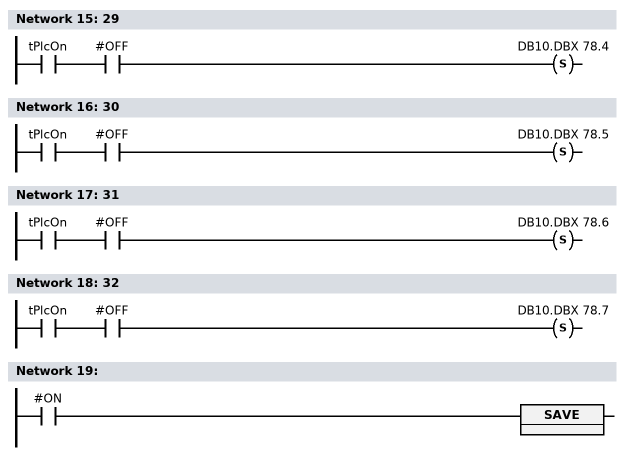
[picture p213: Errors_017-032_GEN2 networks 15-19]
NETWORK
TITLE = 29
      A     "tPlcOn";
      A     #OFF;
      S     DB10.DBX 78.4;
NETWORK
TITLE = 30
      A     "tPlcOn";
      A     #OFF;
      S     DB10.DBX 78.5;
NETWORK
TITLE = 31
      A     "tPlcOn";
      A     #OFF;
      S     DB10.DBX 78.6;
NETWORK
TITLE = 32
      A     "tPlcOn";
      A     #OFF;
      S     DB10.DBX 78.7;
NETWORK
TITLE =
      A     #ON;
      SAVE;
END_FUNCTION

FUNCTION "Errors_033-048_NET" : VOID	// FC 44
TITLE = Errors NET
VERSION : 0.1
VAR_TEMP
  ON : BOOL ;
  OFF : BOOL ;
  tmp_value : INT ;
END_VAR
BEGIN
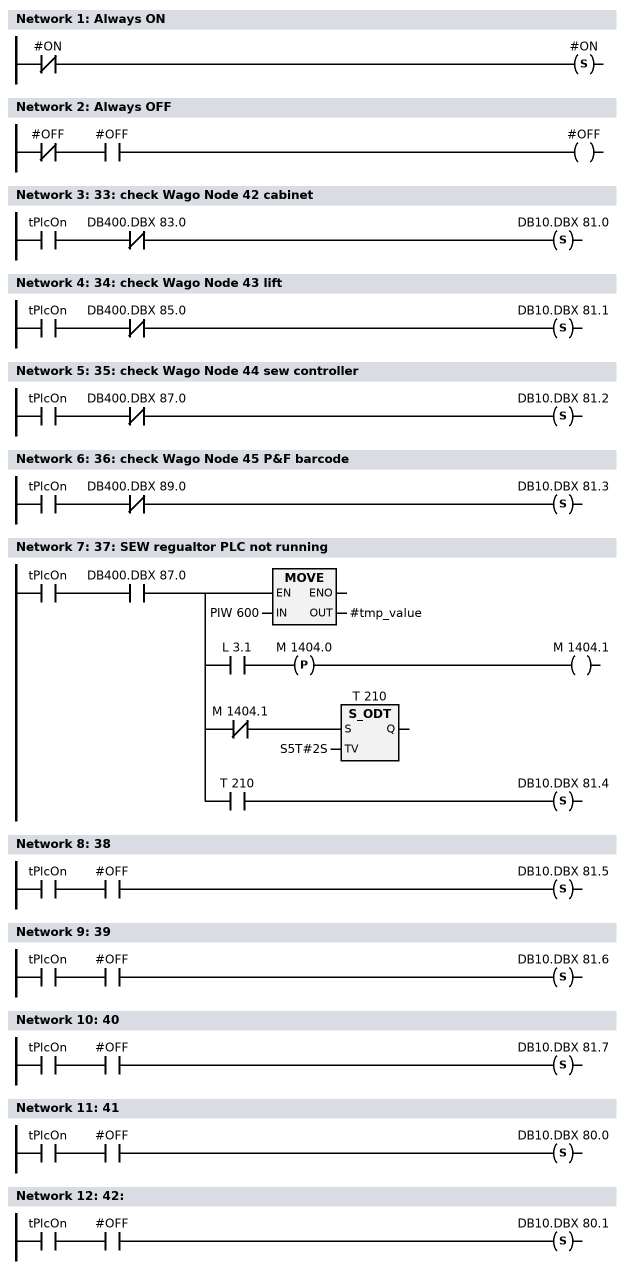
NETWORK
TITLE = Always ON
      AN    #ON;
      S     #ON;
NETWORK
TITLE = Always OFF
      AN    #OFF;
      A     #OFF;
      =     #OFF;
NETWORK
TITLE = 33: check Wago Node 42 cabinet
      A     "tPlcOn";
      AN    DB400.DBX 83.0;
      S     DB10.DBX 81.0;
NETWORK
TITLE = 34: check Wago Node 43 lift
      A     "tPlcOn";
      AN    DB400.DBX 85.0;
      S     DB10.DBX 81.1;
NETWORK
TITLE = 35: check Wago Node 44 sew controller
      A     "tPlcOn";
      AN    DB400.DBX 87.0;
      S     DB10.DBX 81.2;
NETWORK
TITLE = 36: check Wago Node 45 P&F barcode
      A     "tPlcOn";
      AN    DB400.DBX 89.0;
      S     DB10.DBX 81.3;
NETWORK
TITLE = 37: SEW regualtor PLC not running
      A     "tPlcOn";
      A     DB400.DBX 87.0;
      =     L 4.0;
      A     L 4.0;
      JNB   _001;
      L     PIW 600;
      T     #tmp_value;
_001: NOP   0;
      A     L 4.0;
      A     L 3.1;
      FP    M 1404.0;
      =     M 1404.1;
      A     L 4.0;
      AN    M 1404.1;
      L     S5T#2S;
      SD    T 210;
      NOP   0;
      NOP   0;
      NOP   0;
      NOP   0;
      A     L 4.0;
      A     T 210;
      S     DB10.DBX 81.4;
NETWORK
TITLE = 38
      A     "tPlcOn";
      A     #OFF;
      S     DB10.DBX 81.5;
NETWORK
TITLE = 39
      A     "tPlcOn";
      A     #OFF;
      S     DB10.DBX 81.6;
NETWORK
TITLE = 40
      A     "tPlcOn";
      A     #OFF;
      S     DB10.DBX 81.7;
NETWORK
TITLE = 41
      A     "tPlcOn";
      A     #OFF;
      S     DB10.DBX 80.0;
NETWORK
TITLE = 42:
      A     "tPlcOn";
      A     #OFF;
      S     DB10.DBX 80.1;
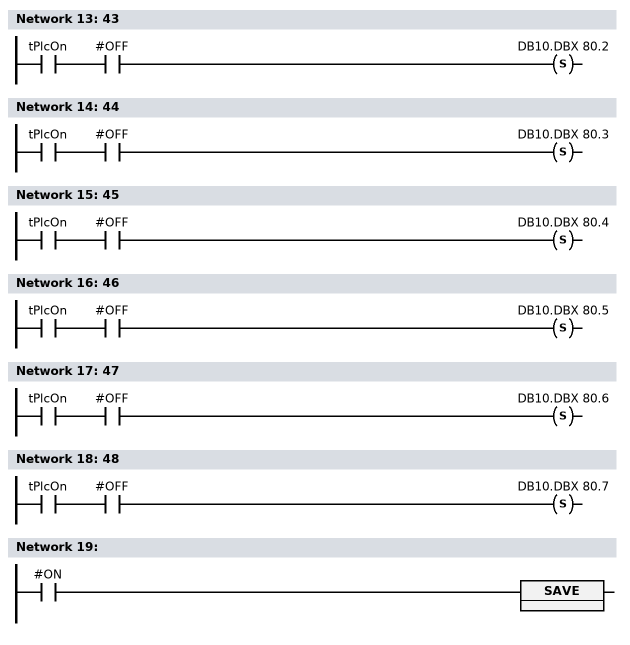
NETWORK
TITLE = 43
      A     "tPlcOn";
      A     #OFF;
      S     DB10.DBX 80.2;
NETWORK
TITLE = 44
      A     "tPlcOn";
      A     #OFF;
      S     DB10.DBX 80.3;
NETWORK
TITLE = 45
      A     "tPlcOn";
      A     #OFF;
      S     DB10.DBX 80.4;
NETWORK
TITLE = 46
      A     "tPlcOn";
      A     #OFF;
      S     DB10.DBX 80.5;
NETWORK
TITLE = 47
      A     "tPlcOn";
      A     #OFF;
      S     DB10.DBX 80.6;
NETWORK
TITLE = 48
      A     "tPlcOn";
      A     #OFF;
      S     DB10.DBX 80.7;
NETWORK
TITLE =
      A     #ON;
      SAVE;
END_FUNCTION

FUNCTION "Errors_113-128" : VOID	// FC 45
TITLE = Errors 113 - 128
VERSION : 0.1
VAR_TEMP
  ON : BOOL ;
END_VAR
BEGIN
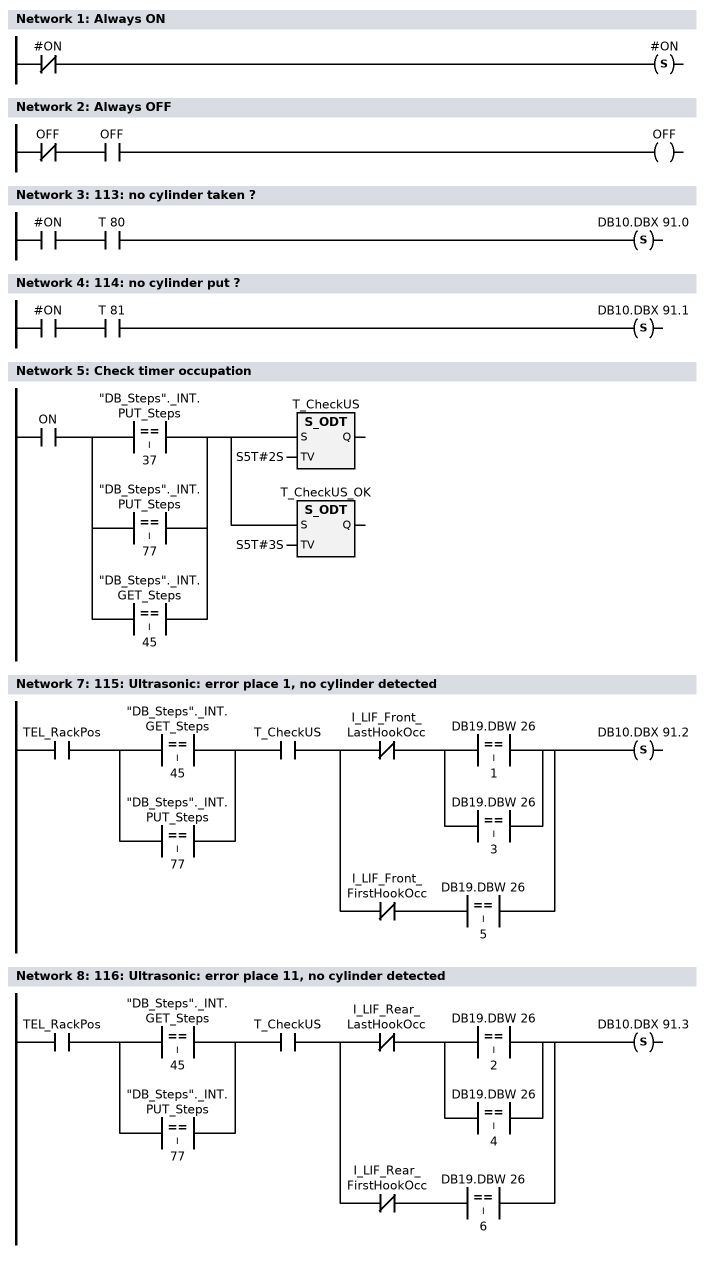
NETWORK
TITLE = Always ON
      AN    #ON;
      S     #ON;
NETWORK
TITLE = Always OFF
      AN    "OFF";
      A     "OFF";
      =     "OFF";
NETWORK
TITLE = 113: no cylinder taken ?
      A     #ON;
      A     T 80;
      S     DB10.DBX 91.0;
NETWORK
TITLE = 114: no cylinder put ?
      A     #ON;
      A     T 81;
      S     DB10.DBX 91.1;
NETWORK
TITLE = Check timer occupation
//T160 time to error
//T161 time to cont
      A     "ON";
      A(;
      O(;
      L     "DB_Steps"._INT.PUT_Steps;
      L     37;
      ==I;
      );
      O(;
      L     "DB_Steps"._INT.PUT_Steps;
      L     77;
      ==I;
      );
      O(;
      L     "DB_Steps"._INT.GET_Steps;
      L     45;
      ==I;
      );
      );
      =     L 1.0;
      A     L 1.0;
      L     S5T#2S;
      SD    "T_CheckUS";
      NOP   0;
      NOP   0;
      NOP   0;
      NOP   0;
      A     L 1.0;
      L     S5T#3S;
      SD    "T_CheckUS_OK";
      NOP   0;
      NOP   0;
      NOP   0;
      NOP   0;
NETWORK
TITLE =
NETWORK
TITLE = 115: Ultrasonic: error place 1, no cylinder detected
      A     "TEL_RackPos";
      A(;
      O(;
      L     "DB_Steps"._INT.GET_Steps;
      L     45;
      ==I;
      );
      O(;
      L     "DB_Steps"._INT.PUT_Steps;
      L     77;
      ==I;
      );
      );
      A     "T_CheckUS";
      A(;
      AN    "I_LIF_Front_LastHookOcc";
      A(;
      O(;
      L     DB19.DBW 26;
      L     1;
      ==I;
      );
      O(;
      L     DB19.DBW 26;
      L     3;
      ==I;
      );
      );
      O;
      AN    "I_LIF_Front_FirstHookOcc";
      A(;
      L     DB19.DBW 26;
      L     5;
      ==I;
      );
      );
      S     DB10.DBX 91.2;
NETWORK
TITLE = 116: Ultrasonic: error place 11, no cylinder detected
      A     "TEL_RackPos";
      A(;
      O(;
      L     "DB_Steps"._INT.GET_Steps;
      L     45;
      ==I;
      );
      O(;
      L     "DB_Steps"._INT.PUT_Steps;
      L     77;
      ==I;
      );
      );
      A     "T_CheckUS";
      A(;
      AN    "I_LIF_Rear_LastHookOcc";
      A(;
      O(;
      L     DB19.DBW 26;
      L     2;
      ==I;
      );
      O(;
      L     DB19.DBW 26;
      L     4;
      ==I;
      );
      );
      O;
      AN    "I_LIF_Rear_FirstHookOcc";
      A(;
      L     DB19.DBW 26;
      L     6;
      ==I;
      );
      );
      S     DB10.DBX 91.3;
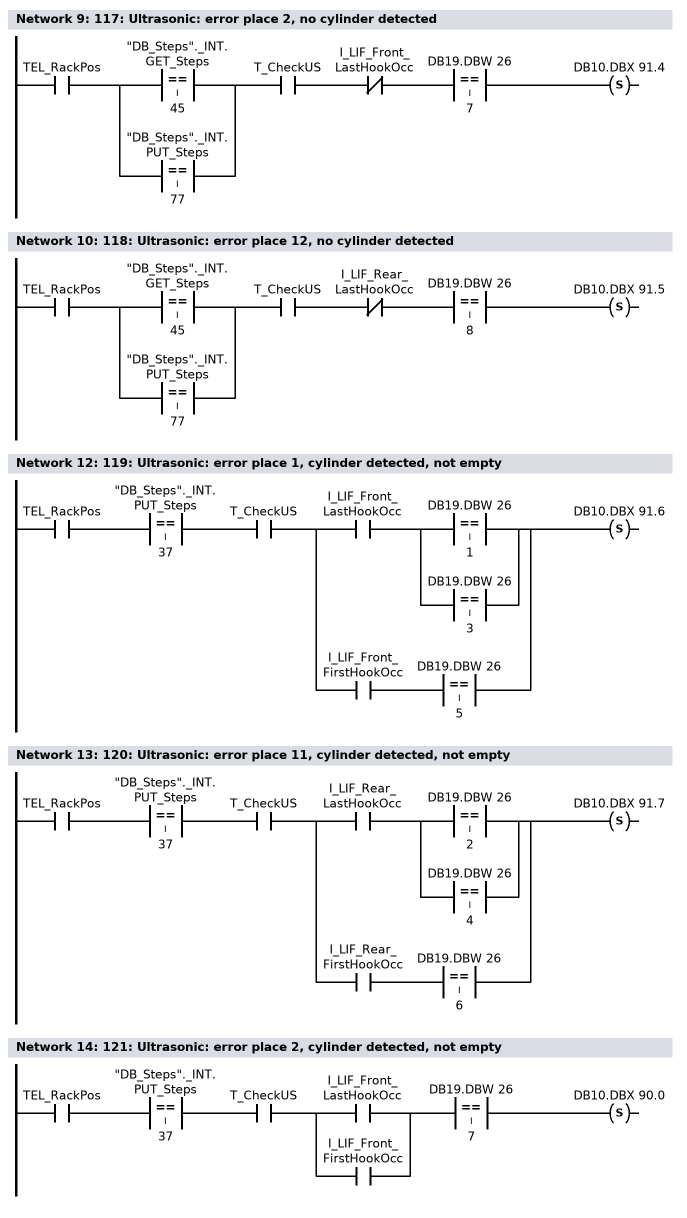
NETWORK
TITLE = 117: Ultrasonic: error place 2, no cylinder detected
      A     "TEL_RackPos";
      A(;
      O(;
      L     "DB_Steps"._INT.GET_Steps;
      L     45;
      ==I;
      );
      O(;
      L     "DB_Steps"._INT.PUT_Steps;
      L     77;
      ==I;
      );
      );
      A     "T_CheckUS";
      AN    "I_LIF_Front_LastHookOcc";
      A(;
      L     DB19.DBW 26;
      L     7;
      ==I;
      );
      S     DB10.DBX 91.4;
NETWORK
TITLE = 118: Ultrasonic: error place 12, no cylinder detected
      A     "TEL_RackPos";
      A(;
      O(;
      L     "DB_Steps"._INT.GET_Steps;
      L     45;
      ==I;
      );
      O(;
      L     "DB_Steps"._INT.PUT_Steps;
      L     77;
      ==I;
      );
      );
      A     "T_CheckUS";
      AN    "I_LIF_Rear_LastHookOcc";
      A(;
      L     DB19.DBW 26;
      L     8;
      ==I;
      );
      S     DB10.DBX 91.5;
NETWORK
TITLE =
NETWORK
TITLE = 119: Ultrasonic: error place 1, cylinder detected, not empty
      A     "TEL_RackPos";
      A(;
      L     "DB_Steps"._INT.PUT_Steps;
      L     37;
      ==I;
      );
      A     "T_CheckUS";
      A(;
      A     "I_LIF_Front_LastHookOcc";
      A(;
      O(;
      L     DB19.DBW 26;
      L     1;
      ==I;
      );
      O(;
      L     DB19.DBW 26;
      L     3;
      ==I;
      );
      );
      O;
      A     "I_LIF_Front_FirstHookOcc";
      A(;
      L     DB19.DBW 26;
      L     5;
      ==I;
      );
      );
      S     DB10.DBX 91.6;
NETWORK
TITLE = 120: Ultrasonic: error place 11, cylinder detected, not empty
      A     "TEL_RackPos";
      A(;
      L     "DB_Steps"._INT.PUT_Steps;
      L     37;
      ==I;
      );
      A     "T_CheckUS";
      A(;
      A     "I_LIF_Rear_LastHookOcc";
      A(;
      O(;
      L     DB19.DBW 26;
      L     2;
      ==I;
      );
      O(;
      L     DB19.DBW 26;
      L     4;
      ==I;
      );
      );
      O;
      A     "I_LIF_Rear_FirstHookOcc";
      A(;
      L     DB19.DBW 26;
      L     6;
      ==I;
      );
      );
      S     DB10.DBX 91.7;
NETWORK
TITLE = 121: Ultrasonic: error place 2, cylinder detected, not empty
      A     "TEL_RackPos";
      A(;
      L     "DB_Steps"._INT.PUT_Steps;
      L     37;
      ==I;
      );
      A     "T_CheckUS";
      A(;
      O     "I_LIF_Front_LastHookOcc";
      O     "I_LIF_Front_FirstHookOcc";
      );
      A(;
      L     DB19.DBW 26;
      L     7;
      ==I;
      );
      S     DB10.DBX 90.0;
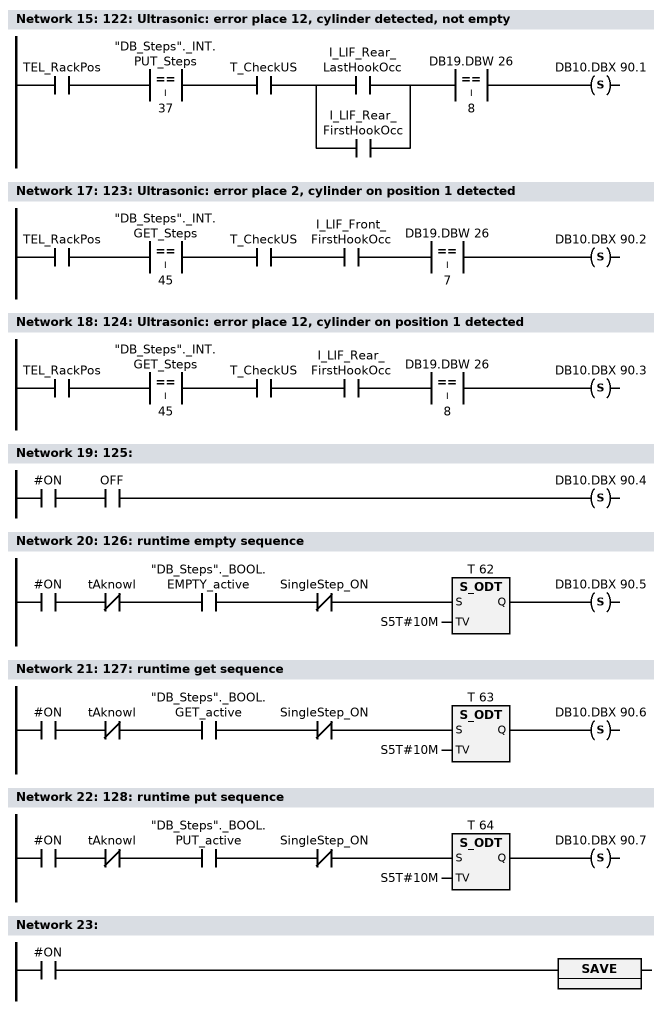
NETWORK
TITLE = 122: Ultrasonic: error place 12, cylinder detected, not empty
      A     "TEL_RackPos";
      A(;
      L     "DB_Steps"._INT.PUT_Steps;
      L     37;
      ==I;
      );
      A     "T_CheckUS";
      A(;
      O     "I_LIF_Rear_LastHookOcc";
      O     "I_LIF_Rear_FirstHookOcc";
      );
      A(;
      L     DB19.DBW 26;
      L     8;
      ==I;
      );
      S     DB10.DBX 90.1;
NETWORK
TITLE =
NETWORK
TITLE = 123: Ultrasonic: error place 2, cylinder on position 1 detected
      A     "TEL_RackPos";
      A(;
      L     "DB_Steps"._INT.GET_Steps;
      L     45;
      ==I;
      );
      A     "T_CheckUS";
      A     "I_LIF_Front_FirstHookOcc";
      A(;
      L     DB19.DBW 26;
      L     7;
      ==I;
      );
      S     DB10.DBX 90.2;
NETWORK
TITLE = 124: Ultrasonic: error place 12, cylinder on position 1 detected
      A     "TEL_RackPos";
      A(;
      L     "DB_Steps"._INT.GET_Steps;
      L     45;
      ==I;
      );
      A     "T_CheckUS";
      A     "I_LIF_Rear_FirstHookOcc";
      A(;
      L     DB19.DBW 26;
      L     8;
      ==I;
      );
      S     DB10.DBX 90.3;
NETWORK
TITLE = 125:
      A     #ON;
      A     "OFF";
      S     DB10.DBX 90.4;
NETWORK
TITLE = 126: runtime empty sequence
      A     #ON;
      AN    "tAknowl";
      A     "DB_Steps"._BOOL.EMPTY_active;
      AN    "SingleStep_ON";
      L     S5T#10M;
      SD    T 62;
      NOP   0;
      NOP   0;
      NOP   0;
      A     T 62;
      S     DB10.DBX 90.5;
NETWORK
TITLE = 127: runtime get sequence
      A     #ON;
      AN    "tAknowl";
      A     "DB_Steps"._BOOL.GET_active;
      AN    "SingleStep_ON";
      L     S5T#10M;
      SD    T 63;
      NOP   0;
      NOP   0;
      NOP   0;
      A     T 63;
      S     DB10.DBX 90.6;
NETWORK
TITLE = 128: runtime put sequence
      A     #ON;
      AN    "tAknowl";
      A     "DB_Steps"._BOOL.PUT_active;
      AN    "SingleStep_ON";
      L     S5T#10M;
      SD    T 64;
      NOP   0;
      NOP   0;
      NOP   0;
      A     T 64;
      S     DB10.DBX 90.7;
NETWORK
TITLE =
      A     #ON;
      SAVE;
END_FUNCTION

FUNCTION "Errors_129-144_08" : VOID	// FC 46
TITLE = Errors
VERSION : 0.1
VAR_TEMP
  ON : BOOL ;
  OFF : BOOL ;
END_VAR
BEGIN
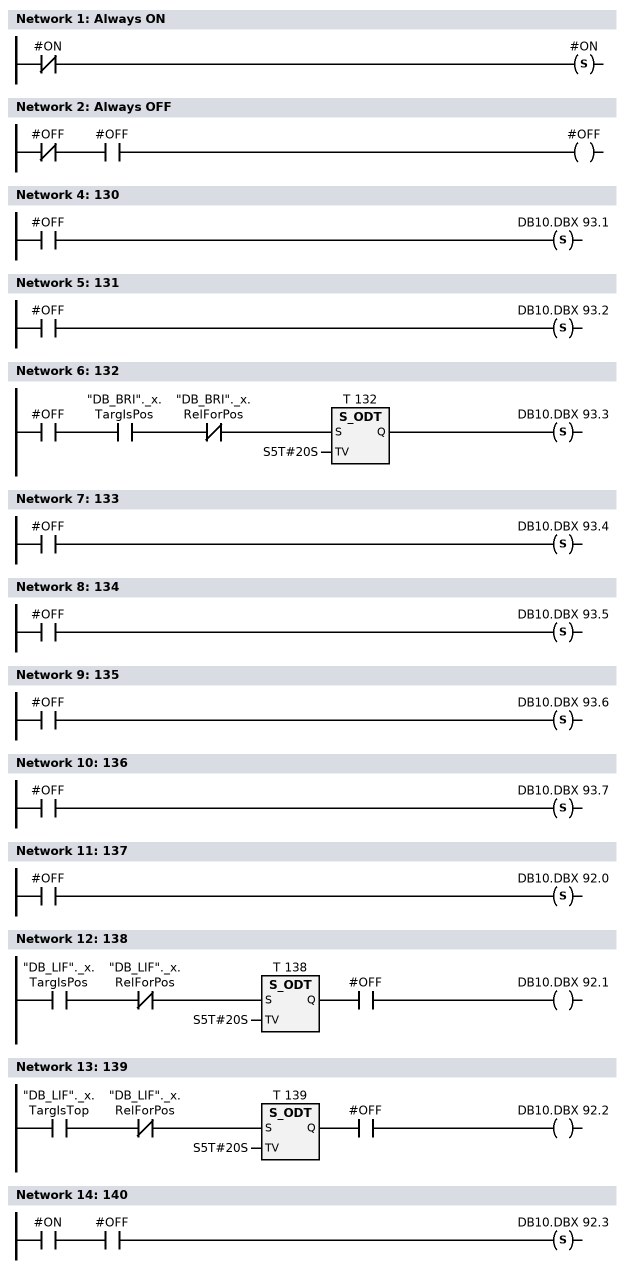
NETWORK
TITLE = Always ON
      AN    #ON;
      S     #ON;
NETWORK
TITLE = Always OFF
      AN    #OFF;
      A     #OFF;
      =     #OFF;
NETWORK
TITLE = 129
//00 in Steps_PUT/NW65
NETWORK
TITLE = 130
//01
      A     #OFF;
      S     DB10.DBX 93.1;
NETWORK
TITLE = 131
//02
      A     #OFF;
      S     DB10.DBX 93.2;
NETWORK
TITLE = 132
//Brücke keine Freigabe für Positionierung
      A     #OFF;
      A     "DB_BRI"._x.TargIsPos;
      AN    "DB_BRI"._x.RelForPos;
      L     S5T#20S;
      SD    T 132;
      NOP   0;
      NOP   0;
      NOP   0;
      A     T 132;
      S     DB10.DBX 93.3;
NETWORK
TITLE = 133
//04
      A     #OFF;
      S     DB10.DBX 93.4;
NETWORK
TITLE = 134
//05
      A     #OFF;
      S     DB10.DBX 93.5;
NETWORK
TITLE = 135
//06
      A     #OFF;
      S     DB10.DBX 93.6;
NETWORK
TITLE = 136
//07
      A     #OFF;
      S     DB10.DBX 93.7;
NETWORK
TITLE = 137
//08
      A     #OFF;
      S     DB10.DBX 92.0;
NETWORK
TITLE = 138
//Lift keine Freigabe für Positionierung
      A(;
      A     "DB_LIF"._x.TargIsPos;
      AN    "DB_LIF"._x.RelForPos;
      L     S5T#20S;
      SD    T 138;
      NOP   0;
      NOP   0;
      NOP   0;
      A     T 138;
      );
      A     #OFF;
      =     DB10.DBX 92.1;
NETWORK
TITLE = 139
//Lift keine Freigabe für Positionierung
      A(;
      A     "DB_LIF"._x.TargIsTop;
      AN    "DB_LIF"._x.RelForPos;
      L     S5T#20S;
      SD    T 139;
      NOP   0;
      NOP   0;
      NOP   0;
      A     T 139;
      );
      A     #OFF;
      =     DB10.DBX 92.2;
NETWORK
TITLE = 140
//Messung Umfang nicht erfolgreich
      A     #ON;
      A     #OFF;
      S     DB10.DBX 92.3;
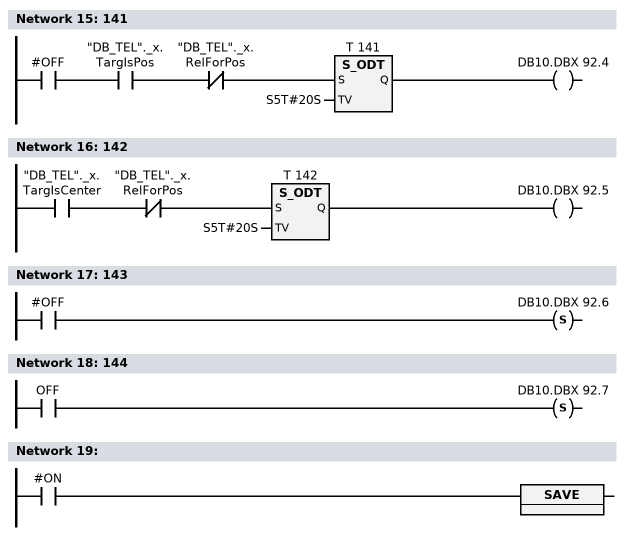
NETWORK
TITLE = 141
//Teleskope keine Freigabe für Positionierung
      A     #OFF;
      A     "DB_TEL"._x.TargIsPos;
      AN    "DB_TEL"._x.RelForPos;
      L     S5T#20S;
      SD    T 141;
      NOP   0;
      NOP   0;
      NOP   0;
      A     T 141;
      =     DB10.DBX 92.4;
NETWORK
TITLE = 142
//Teleskope keine Freigabe für Positionierung
      A     "DB_TEL"._x.TargIsCenter;
      AN    "DB_TEL"._x.RelForPos;
      L     S5T#20S;
      SD    T 142;
      NOP   0;
      NOP   0;
      NOP   0;
      A     T 142;
      =     DB10.DBX 92.5;
NETWORK
TITLE = 143
      A     #OFF;
      S     DB10.DBX 92.6;
NETWORK
TITLE = 144
      A     "OFF";
      S     DB10.DBX 92.7;
NETWORK
TITLE =
      A     #ON;
      SAVE;
END_FUNCTION

FUNCTION "Errors_145-160" : VOID	// FC 47
TITLE = Messages 145 - 160
VERSION : 0.1
VAR_TEMP
  ON : BOOL ;
  OFF : BOOL ;
END_VAR
BEGIN
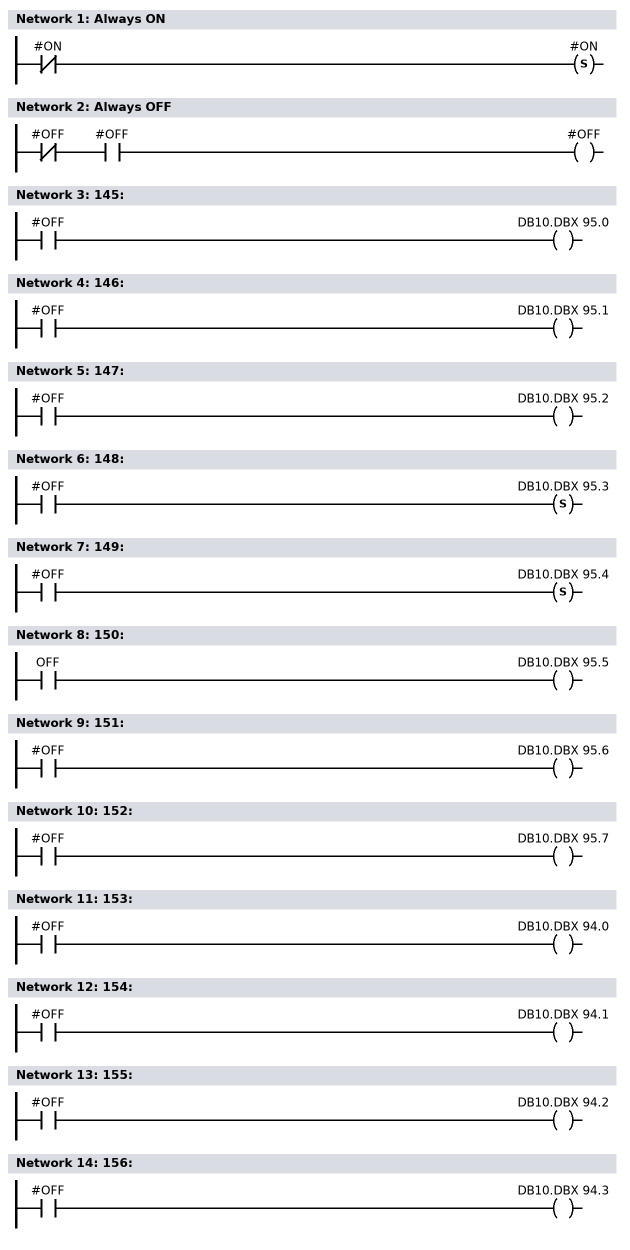
NETWORK
TITLE = Always ON
      AN    #ON;
      S     #ON;
NETWORK
TITLE = Always OFF
      AN    #OFF;
      A     #OFF;
      =     #OFF;
NETWORK
TITLE = 145:
//keine Freigabe Teleskop Fach 1 (Fachtyp)
      A     #OFF;
      =     DB10.DBX 95.0;
NETWORK
TITLE = 146:
//keine Freigabe Teleskop Fach 2 (Fachtyp)
      A     #OFF;
      =     DB10.DBX 95.1;
NETWORK
TITLE = 147:
//keine Freigabe Teleskop Ladestation 1
      A     #OFF;
      =     DB10.DBX 95.2;
NETWORK
TITLE = 148:
//keine Freigabe Teleskop Ladestation 2
      A     #OFF;
      S     DB10.DBX 95.3;
NETWORK
TITLE = 149:
//keine Freigabe Teleskop Ladestation 3
      A     #OFF;
      S     DB10.DBX 95.4;
NETWORK
TITLE = 150:
      A     "OFF";
      =     DB10.DBX 95.5;
NETWORK
TITLE = 151:
      A     #OFF;
      =     DB10.DBX 95.6;
NETWORK
TITLE = 152:
      A     #OFF;
      =     DB10.DBX 95.7;
NETWORK
TITLE = 153:
      A     #OFF;
      =     DB10.DBX 94.0;
NETWORK
TITLE = 154:
      A     #OFF;
      =     DB10.DBX 94.1;
NETWORK
TITLE = 155:
      A     #OFF;
      =     DB10.DBX 94.2;
NETWORK
TITLE = 156:
      A     #OFF;
      =     DB10.DBX 94.3;
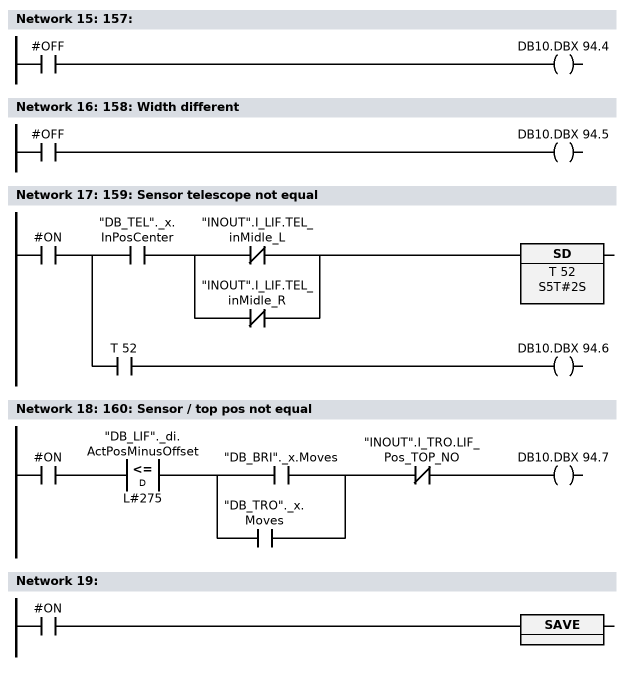
NETWORK
TITLE = 157:
      A     #OFF;
      =     DB10.DBX 94.4;
NETWORK
TITLE = 158: Width different
      A     #OFF;
      =     DB10.DBX 94.5;
NETWORK
TITLE = 159: Sensor telescope not equal
      A     #ON;
      =     L 1.0;
      A     L 1.0;
      A     "DB_TEL"._x.InPosCenter;
      A(;
      ON    "INOUT".I_LIF.TEL_inMidle_L;
      ON    "INOUT".I_LIF.TEL_inMidle_R;
      );
      L     S5T#2S;
      SD    T 52;
      A     L 1.0;
      A     T 52;
      =     DB10.DBX 94.6;
NETWORK
TITLE = 160: Sensor / top pos not equal
      A     #ON;
      A(;
      L     "DB_LIF"._di.ActPosMinusOffset;
      L     L#275;
      <=D;
      );
      A(;
      O     "DB_BRI"._x.Moves;
      O     "DB_TRO"._x.Moves;
      );
      AN    "INOUT".I_TRO.LIF_Pos_TOP_NO;
      =     DB10.DBX 94.7;
NETWORK
TITLE =
      A     #ON;
      SAVE;
END_FUNCTION

FUNCTION "EOff_MachineOff" : VOID	// FC 48
TITLE = EOff Machine off
//TODO disable the remote in auto
VERSION : 0.1
VAR_TEMP
  INT_DivEoff : BOOL ;
  INT_Err_GEN1 : BOOL ;
  INT_Err_GEN2 : BOOL ;
  INT_Err_NET : BOOL ;
  INT_Err_BRI : BOOL ;
  INT_Err_TRO : BOOL ;
  INT_Err_LIF : BOOL ;
  INT_Err_TEL : BOOL ;
  INT_Warn : BOOL ;
  INT_OPM1 : BOOL ;
  INT_OPM2 : BOOL ;
  INT_ERR_06 : BOOL ;
  INT_ERR_07 : BOOL ;
  INT_ERR_08 : BOOL ;
  INT_ERR_09 : BOOL ;
  INT_ERR_10 : BOOL ;
  INT_ERR_11 : BOOL ;
  INT_MSG_01 : BOOL ;
  INT_MSG_02 : BOOL ;
  INT_MSG_03 : BOOL ;
  INT_MSG_04 : BOOL ;
  ON : BOOL ;
  OFF : BOOL ;
END_VAR
BEGIN
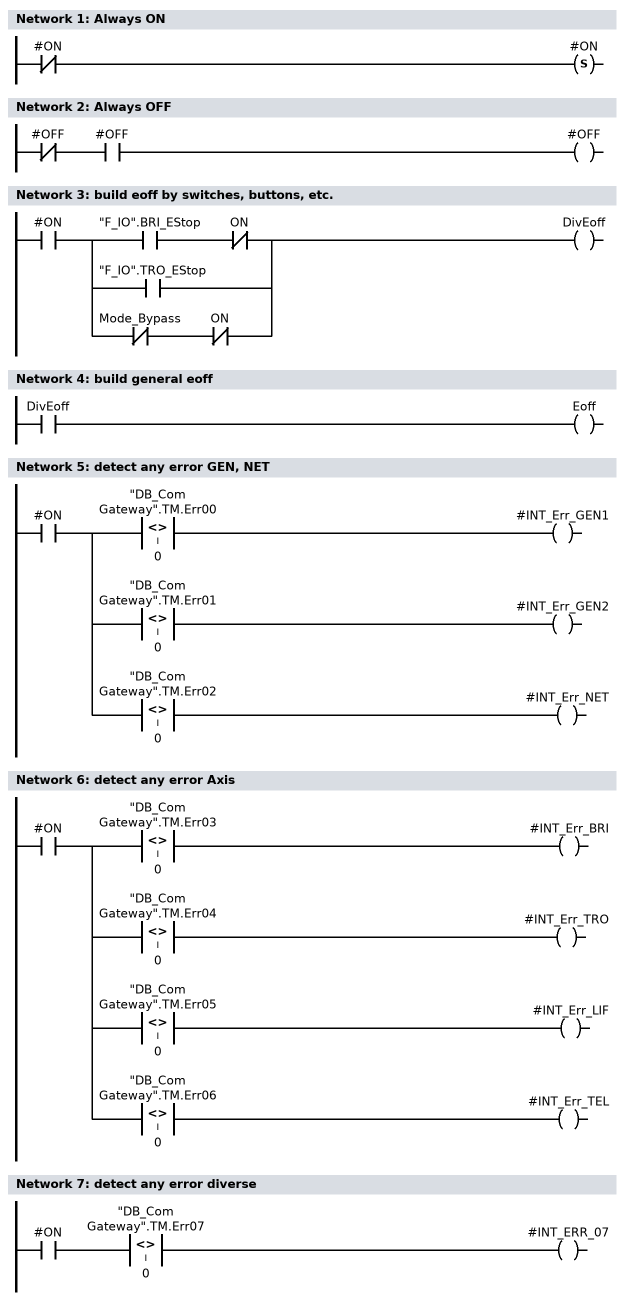
NETWORK
TITLE = Always ON
      AN    #ON;
      S     #ON;
NETWORK
TITLE = Always OFF
      AN    #OFF;
      A     #OFF;
      =     #OFF;
NETWORK
TITLE = build eoff by switches, buttons, etc.
      A     #ON;
      A(;
      A     "F_IO".BRI_EStop;
      AN    "ON";
      O     "F_IO".TRO_EStop;
      O;
      AN    "Mode_Bypass";
      AN    "ON";
      );
      =     "DivEoff";
NETWORK
TITLE = build general eoff
      A     "DivEoff";
      =     "Eoff";
NETWORK
TITLE = detect any error GEN, NET
      A     #ON;
      =     L 3.0;
      A     L 3.0;
      A(;
      L     "DB_ComGateway".TM.Err00;
      L     0;
      <>I;
      );
      =     #INT_Err_GEN1;
      A     L 3.0;
      A(;
      L     "DB_ComGateway".TM.Err01;
      L     0;
      <>I;
      );
      =     #INT_Err_GEN2;
      A     L 3.0;
      A(;
      L     "DB_ComGateway".TM.Err02;
      L     0;
      <>I;
      );
      =     #INT_Err_NET;
NETWORK
TITLE = detect any error Axis
      A     #ON;
      =     L 3.0;
      A     L 3.0;
      A(;
      L     "DB_ComGateway".TM.Err03;
      L     0;
      <>I;
      );
      =     #INT_Err_BRI;
      A     L 3.0;
      A(;
      L     "DB_ComGateway".TM.Err04;
      L     0;
      <>I;
      );
      =     #INT_Err_TRO;
      A     L 3.0;
      A(;
      L     "DB_ComGateway".TM.Err05;
      L     0;
      <>I;
      );
      =     #INT_Err_LIF;
      A     L 3.0;
      A(;
      L     "DB_ComGateway".TM.Err06;
      L     0;
      <>I;
      );
      =     #INT_Err_TEL;
NETWORK
TITLE = detect any error diverse
      A     #ON;
      A(;
      L     "DB_ComGateway".TM.Err07;
      L     0;
      <>I;
      );
      =     #INT_ERR_07;
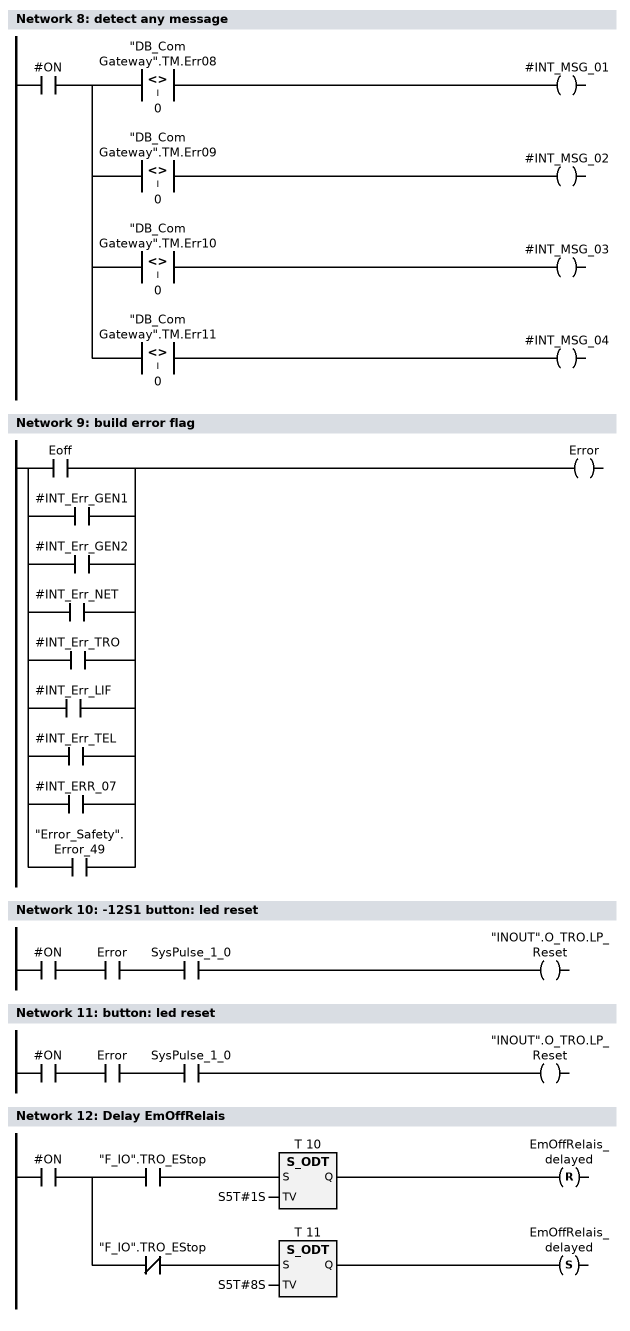
NETWORK
TITLE = detect any message
      A     #ON;
      =     L 3.0;
      A     L 3.0;
      A(;
      L     "DB_ComGateway".TM.Err08;
      L     0;
      <>I;
      );
      =     #INT_MSG_01;
      A     L 3.0;
      A(;
      L     "DB_ComGateway".TM.Err09;
      L     0;
      <>I;
      );
      =     #INT_MSG_02;
      A     L 3.0;
      A(;
      L     "DB_ComGateway".TM.Err10;
      L     0;
      <>I;
      );
      =     #INT_MSG_03;
      A     L 3.0;
      A(;
      L     "DB_ComGateway".TM.Err11;
      L     0;
      <>I;
      );
      =     #INT_MSG_04;
NETWORK
TITLE = build error flag
//xOff for error words
//
      O     "Eoff";
      O     #INT_Err_GEN1;
      O     #INT_Err_GEN2;
      O     #INT_Err_NET;
      O     #INT_Err_TRO;
      O     #INT_Err_LIF;
      O     #INT_Err_TEL;
      O     #INT_ERR_07;
      O     "Error_Safety".Error_49;
      =     "Error";
NETWORK
TITLE = -12S1 button: led reset
      A     #ON;
      A     "Error";
      A     "SysPulse_1_0";
      =     "INOUT".O_TRO.LP_Reset;
NETWORK
TITLE = button: led reset
      A     #ON;
      A     "Error";
      A     "SysPulse_1_0";
      =     "INOUT".O_TRO.LP_Reset;
NETWORK
TITLE = Delay EmOffRelais
      A     #ON;
      =     L 3.0;
      A     L 3.0;
      A     "F_IO".TRO_EStop;
      L     S5T#1S;
      SD    T 10;
      NOP   0;
      NOP   0;
      NOP   0;
      A     T 10;
      R     "EmOffRelais_delayed";
      A     L 3.0;
      AN    "F_IO".TRO_EStop;
      L     S5T#8S;
      SD    T 11;
      NOP   0;
      NOP   0;
      NOP   0;
      A     T 11;
      S     "EmOffRelais_delayed";
END_FUNCTION

FUNCTION "OP_Mode" : VOID	// FC 49
TITLE = OP Mode
//Sicherheitsbaugruppen noch nicht in Betrieb !!!
VERSION : 0.1
VAR_TEMP
  TEMP_DINT_00 : DINT ;
  TEMP_DINT_01 : DINT ;
  TEMP_BOOL_00 : BOOL ;
  TEMP_BOOL_01 : BOOL ;
  TEMP_BOOL_02 : BOOL ;
  TEMP_BOOL_03 : BOOL ;
  TEMP_BOOL_04 : BOOL ;
  TEMP_BOOL_05 : BOOL ;
  TEMP_BOOL_06 : BOOL ;
  value : INT ;
  lampPrio : INT ;
  ON : BOOL ;
  OFF : BOOL ;
  delay : BOOL ;
END_VAR
BEGIN
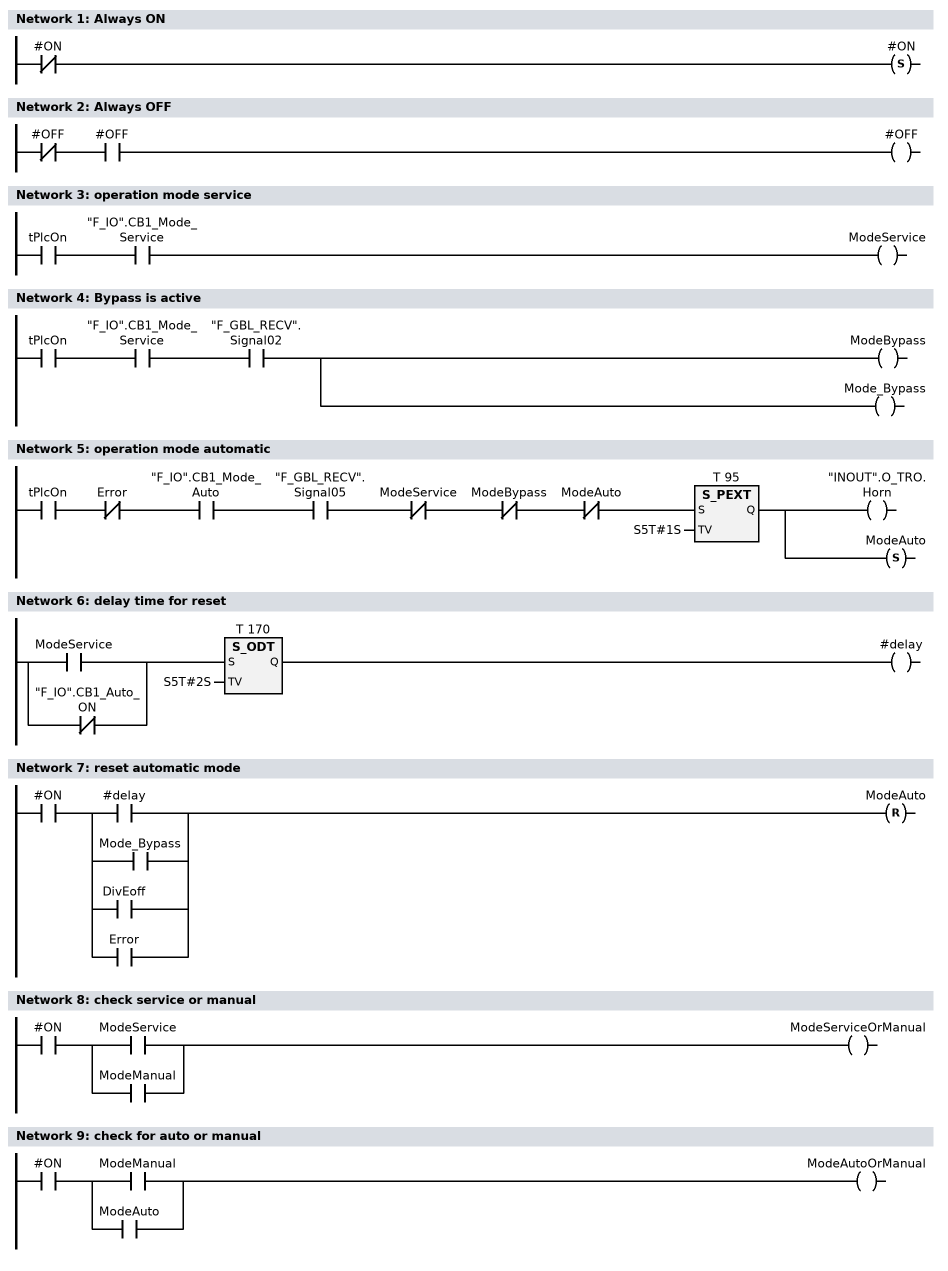
NETWORK
TITLE = Always ON
      AN    #ON;
      S     #ON;
NETWORK
TITLE = Always OFF
      AN    #OFF;
      A     #OFF;
      =     #OFF;
NETWORK
TITLE = operation mode service
      A     "tPlcOn";
      A     "F_IO".CB1_Mode_Service;
      =     "ModeService";
NETWORK
TITLE = Bypass is active
      A     "tPlcOn";
      A     "F_IO".CB1_Mode_Service;
      A     "F_GBL_RECV".Signal02;
      =     "ModeBypass";
      =     "Mode_Bypass";
NETWORK
TITLE = operation mode automatic
      A     "tPlcOn";
      AN    "Error";
      A     "F_IO".CB1_Mode_Auto;
      A     "F_GBL_RECV".Signal05;
      AN    "ModeService";
      AN    "ModeBypass";
      AN    "ModeAuto";
      L     S5T#1S;
      SE    T 95;
      NOP   0;
      NOP   0;
      NOP   0;
      A     T 95;
      =     "INOUT".O_TRO.Horn;
      S     "ModeAuto";
NETWORK
TITLE = delay time for reset
      A(;
      O     "ModeService";
      ON    "F_IO".CB1_Auto_ON;
      );
      L     S5T#2S;
      SD    T 170;
      NOP   0;
      NOP   0;
      NOP   0;
      A     T 170;
      =     #delay;
NETWORK
TITLE = reset automatic mode
      A     #ON;
      A(;
      O     #delay;
      O     "Mode_Bypass";
      O     "DivEoff";
      O     "Error";
      );
      R     "ModeAuto";
NETWORK
TITLE = check service or manual
      A     #ON;
      A(;
      O     "ModeService";
      O     "ModeManual";
      );
      =     "ModeServiceOrManual";
NETWORK
TITLE = check for auto or manual
      A     #ON;
      A(;
      O     "ModeManual";
      O     "ModeAuto";
      );
      =     "ModeAutoOrManual";
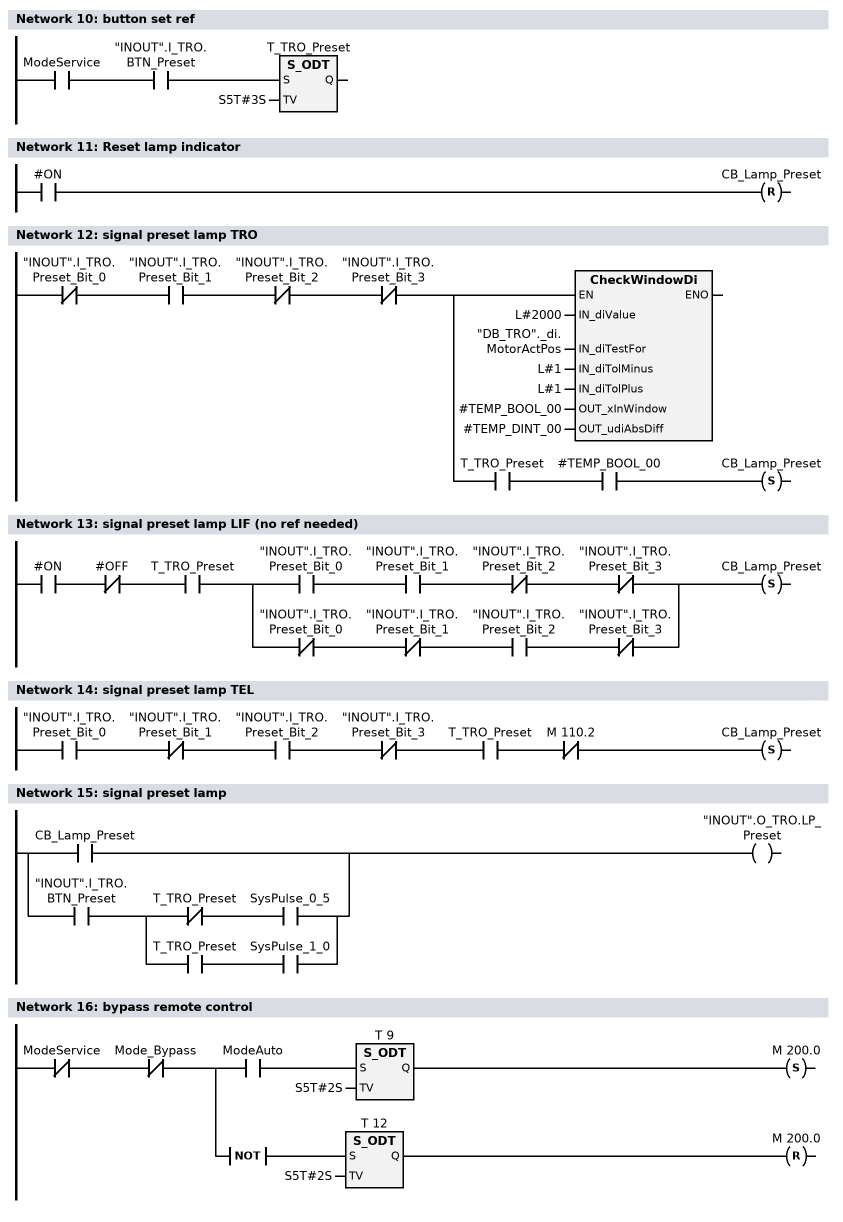
NETWORK
TITLE = button set ref
      A     "ModeService";
      A     "INOUT".I_TRO.BTN_Preset;
      L     S5T#3S;
      SD    "T_TRO_Preset";
      NOP   0;
      NOP   0;
      NOP   0;
      NOP   0;
NETWORK
TITLE = Reset lamp indicator
      A     #ON;
      R     "CB_Lamp_Preset";
NETWORK
TITLE = signal preset lamp TRO
      AN    "INOUT".I_TRO.Preset_Bit_0;
      A     "INOUT".I_TRO.Preset_Bit_1;
      AN    "INOUT".I_TRO.Preset_Bit_2;
      AN    "INOUT".I_TRO.Preset_Bit_3;
      =     L 15.0;
      A     L 15.0;
      JNB   _001;
      CALL  "CheckWindowDi" (
           IN_diValue               := L#2000,
           IN_diTestFor             := "DB_TRO"._di.MotorActPos,
           IN_diTolMinus            := L#1,
           IN_diTolPlus             := L#1,
           OUT_xInWindow            := #TEMP_BOOL_00,
           OUT_udiAbsDiff           := #TEMP_DINT_00);
_001: NOP   0;
      A     L 15.0;
      A     "T_TRO_Preset";
      A     #TEMP_BOOL_00;
      S     "CB_Lamp_Preset";
NETWORK
TITLE = signal preset lamp LIF (no ref needed)
      A     #ON;
      AN    #OFF;
      A     "T_TRO_Preset";
      A(;
      A     "INOUT".I_TRO.Preset_Bit_0;
      A     "INOUT".I_TRO.Preset_Bit_1;
      AN    "INOUT".I_TRO.Preset_Bit_2;
      AN    "INOUT".I_TRO.Preset_Bit_3;
      O;
      AN    "INOUT".I_TRO.Preset_Bit_0;
      AN    "INOUT".I_TRO.Preset_Bit_1;
      A     "INOUT".I_TRO.Preset_Bit_2;
      AN    "INOUT".I_TRO.Preset_Bit_3;
      );
      S     "CB_Lamp_Preset";
NETWORK
TITLE = signal preset lamp TEL
      A     "INOUT".I_TRO.Preset_Bit_0;
      AN    "INOUT".I_TRO.Preset_Bit_1;
      A     "INOUT".I_TRO.Preset_Bit_2;
      AN    "INOUT".I_TRO.Preset_Bit_3;
      A     "T_TRO_Preset";
      AN    M 110.2;
      S     "CB_Lamp_Preset";
NETWORK
TITLE = signal preset lamp
      O     "CB_Lamp_Preset";
      O;
      A     "INOUT".I_TRO.BTN_Preset;
      A(;
      AN    "T_TRO_Preset";
      A     "SysPulse_0_5";
      O;
      A     "T_TRO_Preset";
      A     "SysPulse_1_0";
      );
      =     "INOUT".O_TRO.LP_Preset;
NETWORK
TITLE = bypass remote control
//need to be in safe code
      AN    "ModeService";
      AN    "Mode_Bypass";
      =     L 15.0;
      A     L 15.0;
      A     "ModeAuto";
      L     S5T#2S;
      SD    T 9;
      NOP   0;
      NOP   0;
      NOP   0;
      A     T 9;
      S     M 200.0;
      A     L 15.0;
      NOT;
      L     S5T#2S;
      SD    T 12;
      NOP   0;
      NOP   0;
      NOP   0;
      A     T 12;
      R     M 200.0;
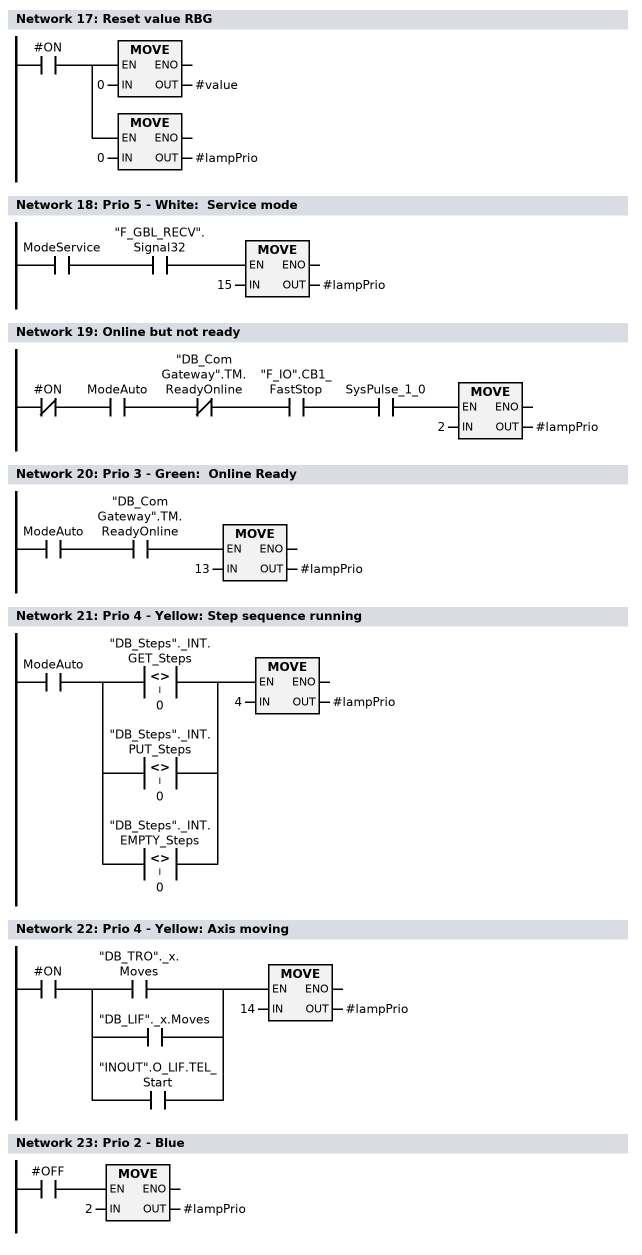
NETWORK
TITLE = Reset value RBG
      A     #ON;
      =     L 15.0;
      A     L 15.0;
      JNB   _002;
      L     0;
      T     #value;
_002: NOP   0;
      A     L 15.0;
      JNB   _003;
      L     0;
      T     #lampPrio;
_003: NOP   0;
NETWORK
TITLE = Prio 5 - White:  Service mode
      A     "ModeService";
      A     "F_GBL_RECV".Signal32;
      JNB   _004;
      L     15;
      T     #lampPrio;
_004: NOP   0;
NETWORK
TITLE = Online but not ready
      AN    #ON;
      A     "ModeAuto";
      AN    "DB_ComGateway".TM.ReadyOnline;
      A     "F_IO".CB1_FastStop;
      A     "SysPulse_1_0";
      JNB   _005;
      L     2;
      T     #lampPrio;
_005: NOP   0;
NETWORK
TITLE = Prio 3 - Green:  Online Ready
      A     "ModeAuto";
      A     "DB_ComGateway".TM.ReadyOnline;
      JNB   _006;
      L     13;
      T     #lampPrio;
_006: NOP   0;
NETWORK
TITLE = Prio 4 - Yellow: Step sequence running
      A     "ModeAuto";
      A(;
      O(;
      L     "DB_Steps"._INT.GET_Steps;
      L     0;
      <>I;
      );
      O(;
      L     "DB_Steps"._INT.PUT_Steps;
      L     0;
      <>I;
      );
      O(;
      L     "DB_Steps"._INT.EMPTY_Steps;
      L     0;
      <>I;
      );
      );
      JNB   _007;
      L     4;
      T     #lampPrio;
_007: NOP   0;
NETWORK
TITLE = Prio 4 - Yellow: Axis moving
      A     #ON;
      A(;
      O     "DB_TRO"._x.Moves;
      O     "DB_LIF"._x.Moves;
      O     "INOUT".O_LIF.TEL_Start;
      );
      JNB   _008;
      L     14;
      T     #lampPrio;
_008: NOP   0;
NETWORK
TITLE = Prio 2 - Blue
      A     #OFF;
      JNB   _009;
      L     2;
      T     #lampPrio;
_009: NOP   0;
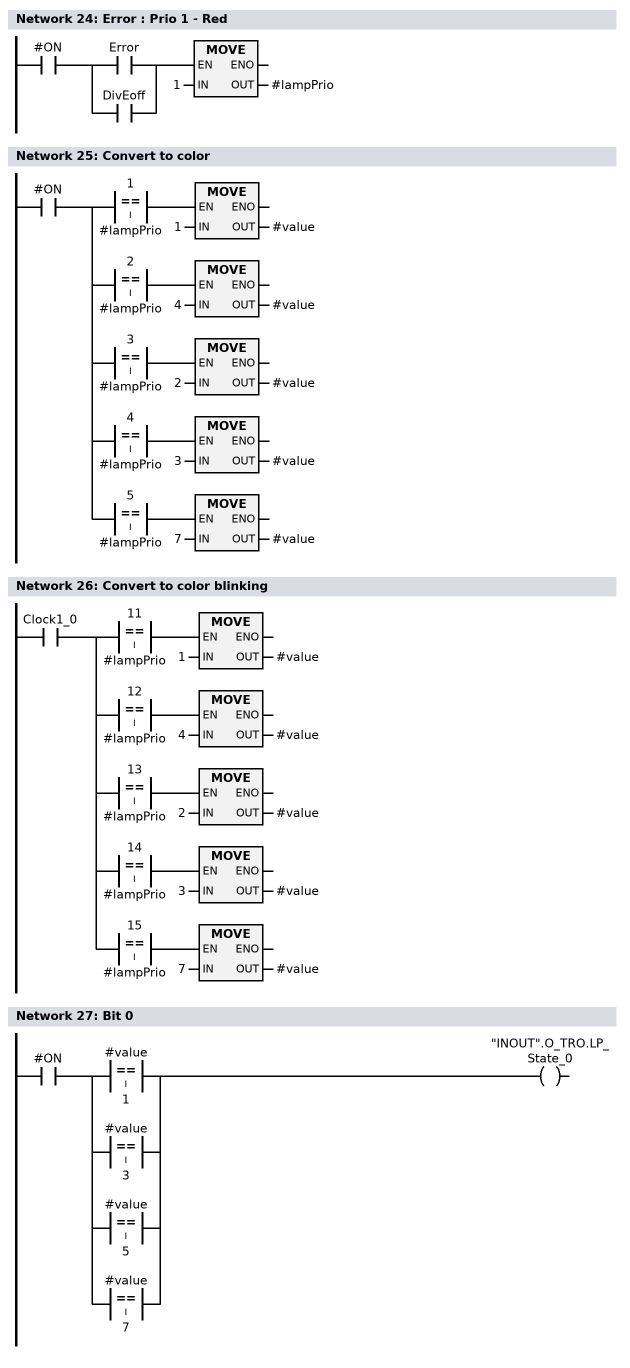
NETWORK
TITLE = Error : Prio 1 - Red
      A     #ON;
      A(;
      O     "Error";
      O     "DivEoff";
      );
      JNB   _00a;
      L     1;
      T     #lampPrio;
_00a: NOP   0;
NETWORK
TITLE = Convert to color
      A     #ON;
      =     L 15.0;
      A     L 15.0;
      A(;
      L     1;
      L     #lampPrio;
      ==I;
      );
      JNB   _00b;
      L     1;
      T     #value;
_00b: NOP   0;
      A     L 15.0;
      A(;
      L     2;
      L     #lampPrio;
      ==I;
      );
      JNB   _00c;
      L     4;
      T     #value;
_00c: NOP   0;
      A     L 15.0;
      A(;
      L     3;
      L     #lampPrio;
      ==I;
      );
      JNB   _00d;
      L     2;
      T     #value;
_00d: NOP   0;
      A     L 15.0;
      A(;
      L     4;
      L     #lampPrio;
      ==I;
      );
      JNB   _00e;
      L     3;
      T     #value;
_00e: NOP   0;
      A     L 15.0;
      A(;
      L     5;
      L     #lampPrio;
      ==I;
      );
      JNB   _00f;
      L     7;
      T     #value;
_00f: NOP   0;
NETWORK
TITLE = Convert to color blinking
      A     "Clock1_0";
      =     L 15.0;
      A     L 15.0;
      A(;
      L     11;
      L     #lampPrio;
      ==I;
      );
      JNB   _010;
      L     1;
      T     #value;
_010: NOP   0;
      A     L 15.0;
      A(;
      L     12;
      L     #lampPrio;
      ==I;
      );
      JNB   _011;
      L     4;
      T     #value;
_011: NOP   0;
      A     L 15.0;
      A(;
      L     13;
      L     #lampPrio;
      ==I;
      );
      JNB   _012;
      L     2;
      T     #value;
_012: NOP   0;
      A     L 15.0;
      A(;
      L     14;
      L     #lampPrio;
      ==I;
      );
      JNB   _013;
      L     3;
      T     #value;
_013: NOP   0;
      A     L 15.0;
      A(;
      L     15;
      L     #lampPrio;
      ==I;
      );
      JNB   _014;
      L     7;
      T     #value;
_014: NOP   0;
NETWORK
TITLE = Bit 0
//BIT 0 1 2 Color
//-----------------
//0    0 0 0 Off
//1    1 0 0 red
//2    0 1 0 green
//3    1 1 0 yellow
//4    0 0 1 blue
//5    1 0 1 viloet 
//6    0 1 1 turque
//7    1 1 1 white
      A     #ON;
      A(;
      O(;
      L     #value;
      L     1;
      ==I;
      );
      O(;
      L     #value;
      L     3;
      ==I;
      );
      O(;
      L     #value;
      L     5;
      ==I;
      );
      O(;
      L     #value;
      L     7;
      ==I;
      );
      );
      =     "INOUT".O_TRO.LP_State_0;
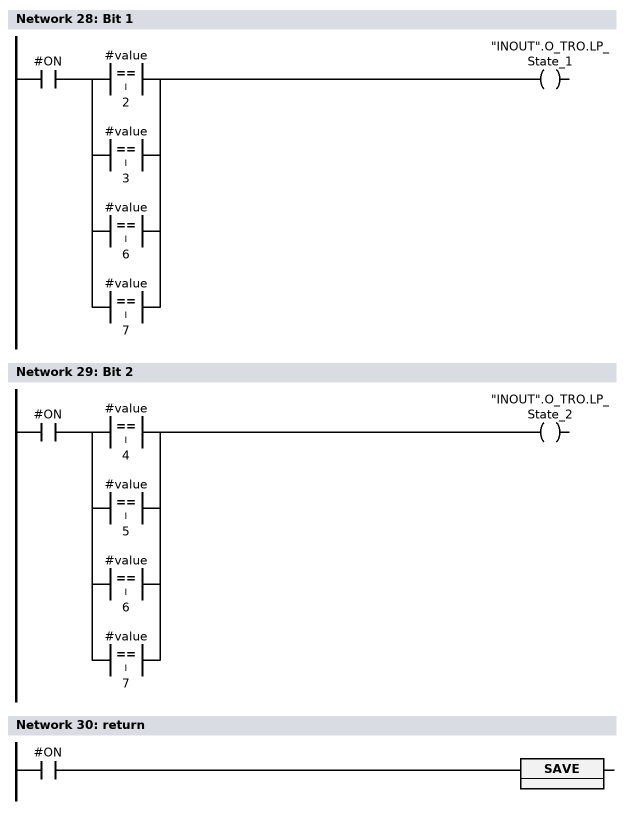
NETWORK
TITLE = Bit 1
      A     #ON;
      A(;
      O(;
      L     #value;
      L     2;
      ==I;
      );
      O(;
      L     #value;
      L     3;
      ==I;
      );
      O(;
      L     #value;
      L     6;
      ==I;
      );
      O(;
      L     #value;
      L     7;
      ==I;
      );
      );
      =     "INOUT".O_TRO.LP_State_1;
NETWORK
TITLE = Bit 2
      A     #ON;
      A(;
      O(;
      L     #value;
      L     4;
      ==I;
      );
      O(;
      L     #value;
      L     5;
      ==I;
      );
      O(;
      L     #value;
      L     6;
      ==I;
      );
      O(;
      L     #value;
      L     7;
      ==I;
      );
      );
      =     "INOUT".O_TRO.LP_State_2;
NETWORK
TITLE = return
      A     #ON;
      SAVE;
END_FUNCTION

FUNCTION "Send_Buffer" : VOID	// FC 52
TITLE = Handle Buffer
VERSION : 0.1
VAR_TEMP
  Count : INT ;
  POINT1 : DWORD ;
  POINT2 : DWORD ;
  POINT3 : DWORD ;
  POINT4 : DWORD ;
  Data : BOOL ;
  Space : BOOL ;
  Loop : INT ;
  Return : INT ;
END_VAR
BEGIN
NETWORK
TITLE = Init values
      L     0;
      T     #Count;
      L     L#52;
      SLD   3;
      T     #POINT1;
      L     L#26;
      SLD   3;
      T     #POINT2;
      OPN   "Moves";
l0:   NOP   0;	// Start of main loop
NETWORK
TITLE = Check for Data
      L     DBW [#POINT1];
      L     0;
      <>I;
      =     #Data;
NETWORK
TITLE = Check for Space
      L     DBW [#POINT2];
      L     0;
      ==I;
      =     #Space;
NETWORK
TITLE = Copy up
      A     #Data;
      A     #Space;
      JCN   m0;
      L     #POINT1;
      T     #POINT3;
      L     #POINT2;
      T     #POINT4;
      L     0;
      T     #Loop;
mm:   L     DBW [#POINT3];
      T     DBW [#POINT4];
      L     0;
      T     DBW [#POINT3];
      L     #POINT3;
      L     L#16;
      +D;
      T     #POINT3;
      L     #POINT4;
      L     L#16;
      +D;
      T     #POINT4;
      L     #Loop;
      L     1;
      +I;
      T     #Loop;
      L     13;
      <I;
      JC    mm;
m0:   NOP   0;
NETWORK
TITLE = Next loop ?
      L     #POINT1;
      SRD   3;
      L     L#26;
      +D;
      SLD   3;
      T     #POINT1;
      L     #POINT2;
      SRD   3;
      L     L#26;
      +D;
      SLD   3;
      T     #POINT2;
      L     #Count;
      L     1;
      +I;
      T     #Count;
      L     49;
      >=I;
      JCN   l0;
NETWORK
TITLE =
      SET;
      SAVE;
END_FUNCTION

FUNCTION "MSG_161-176" : VOID	// FC 55
TITLE = Messages 161 - 176
AUTHOR : Koenig
VERSION : 0.1
VAR_TEMP
  ON : BOOL ;
  OFF : BOOL ;
END_VAR
BEGIN
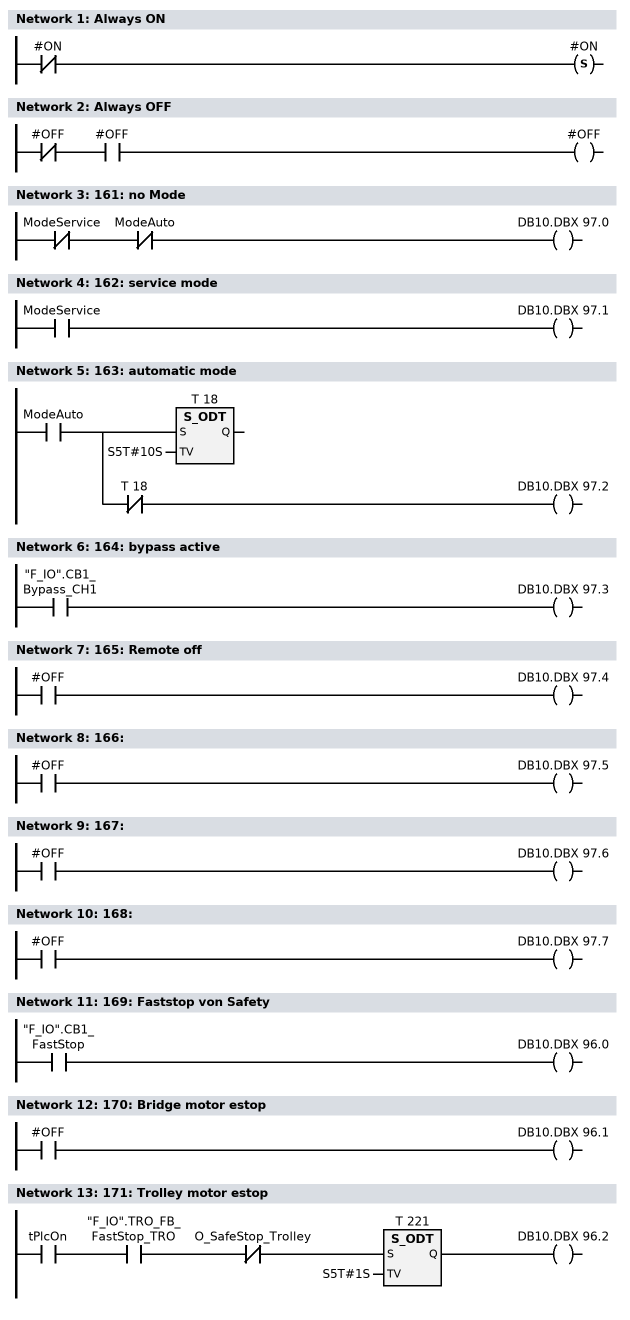
NETWORK
TITLE = Always ON
      AN    #ON;
      S     #ON;
NETWORK
TITLE = Always OFF
      AN    #OFF;
      A     #OFF;
      =     #OFF;
NETWORK
TITLE = 161: no Mode
      AN    "ModeService";
      AN    "ModeAuto";
      =     DB10.DBX 97.0;
NETWORK
TITLE = 162: service mode
      A     "ModeService";
      =     DB10.DBX 97.1;
NETWORK
TITLE = 163: automatic mode
      A     "ModeAuto";
      =     L 1.0;
      A     L 1.0;
      L     S5T#10S;
      SD    T 18;
      NOP   0;
      NOP   0;
      NOP   0;
      NOP   0;
      A     L 1.0;
      AN    T 18;
      =     DB10.DBX 97.2;
NETWORK
TITLE = 164: bypass active
      A     "F_IO".CB1_Bypass_CH1;
      =     DB10.DBX 97.3;
NETWORK
TITLE = 165: Remote off
      A     #OFF;
      =     DB10.DBX 97.4;
NETWORK
TITLE = 166:
      A     #OFF;
      =     DB10.DBX 97.5;
NETWORK
TITLE = 167:
      A     #OFF;
      =     DB10.DBX 97.6;
NETWORK
TITLE = 168:
      A     #OFF;
      =     DB10.DBX 97.7;
NETWORK
TITLE = 169: Faststop von Safety
      A     "F_IO".CB1_FastStop;
      =     DB10.DBX 96.0;
NETWORK
TITLE = 170: Bridge motor estop
      A     #OFF;
      =     DB10.DBX 96.1;
NETWORK
TITLE = 171: Trolley motor estop
      A     "tPlcOn";
      A     "F_IO".TRO_FB_FastStop_TRO;
      AN    "O_SafeStop_Trolley";
      L     S5T#1S;
      SD    T 221;
      NOP   0;
      NOP   0;
      NOP   0;
      A     T 221;
      =     DB10.DBX 96.2;
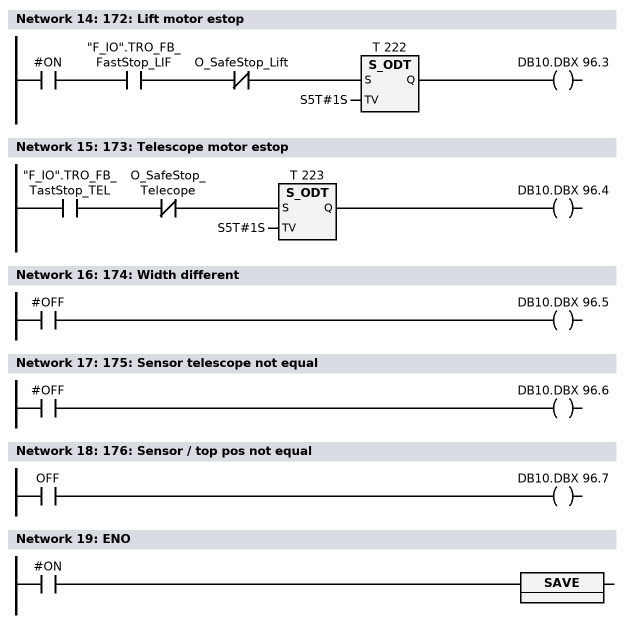
NETWORK
TITLE = 172: Lift motor estop
      A     #ON;
      A     "F_IO".TRO_FB_FastStop_LIF;
      AN    "O_SafeStop_Lift";
      L     S5T#1S;
      SD    T 222;
      NOP   0;
      NOP   0;
      NOP   0;
      A     T 222;
      =     DB10.DBX 96.3;
NETWORK
TITLE = 173: Telescope motor estop
      A     "F_IO".TRO_FB_TastStop_TEL;
      AN    "O_SafeStop_Telecope";
      L     S5T#1S;
      SD    T 223;
      NOP   0;
      NOP   0;
      NOP   0;
      A     T 223;
      =     DB10.DBX 96.4;
NETWORK
TITLE = 174: Width different
      A     #OFF;
      =     DB10.DBX 96.5;
NETWORK
TITLE = 175: Sensor telescope not equal
      A     #OFF;
      =     DB10.DBX 96.6;
NETWORK
TITLE = 176: Sensor / top pos not equal
      A     "OFF";
      =     DB10.DBX 96.7;
NETWORK
TITLE = ENO
      A     #ON;
      SAVE;
END_FUNCTION

FUNCTION "MSG_177_192" : VOID	// FC 56
TITLE = Messages 177 - 192
AUTHOR : Koenig
VERSION : 0.1
VAR_TEMP
  ON : BOOL ;
  OFF : BOOL ;
END_VAR
BEGIN
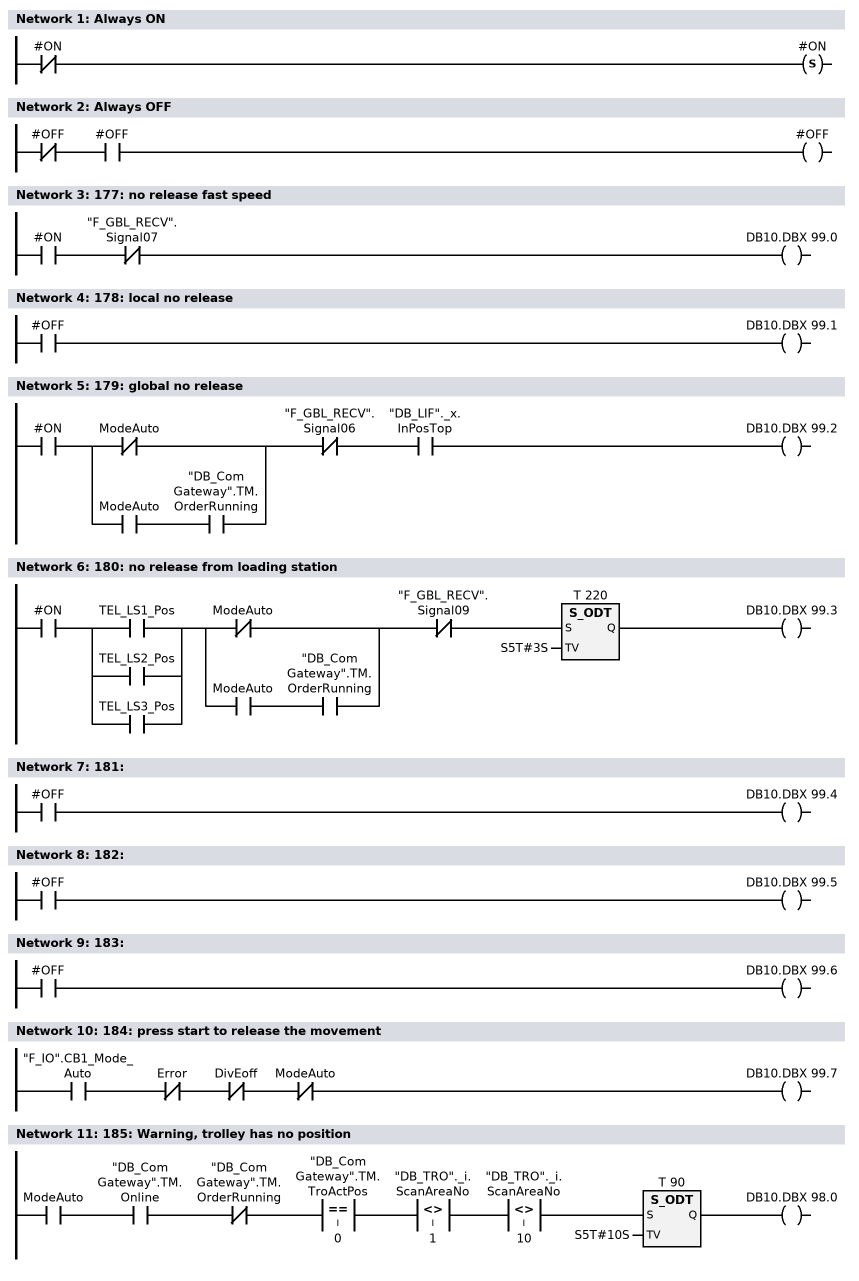
NETWORK
TITLE = Always ON
      AN    #ON;
      S     #ON;
NETWORK
TITLE = Always OFF
      AN    #OFF;
      A     #OFF;
      =     #OFF;
NETWORK
TITLE = 177: no release fast speed
      A     #ON;
      AN    "F_GBL_RECV".Signal07;
      =     DB10.DBX 99.0;
NETWORK
TITLE = 178: local no release
      A     #OFF;
      =     DB10.DBX 99.1;
NETWORK
TITLE = 179: global no release
      A     #ON;
      A(;
      ON    "ModeAuto";
      O;
      A     "ModeAuto";
      A     "DB_ComGateway".TM.OrderRunning;
      );
      AN    "F_GBL_RECV".Signal06;
      A     "DB_LIF"._x.InPosTop;
      =     DB10.DBX 99.2;
NETWORK
TITLE = 180: no release from loading station
      A     #ON;
      A(;
      O     "TEL_LS1_Pos";
      O     "TEL_LS2_Pos";
      O     "TEL_LS3_Pos";
      );
      A(;
      ON    "ModeAuto";
      O;
      A     "ModeAuto";
      A     "DB_ComGateway".TM.OrderRunning;
      );
      AN    "F_GBL_RECV".Signal09;
      L     S5T#3S;
      SD    T 220;
      NOP   0;
      NOP   0;
      NOP   0;
      A     T 220;
      =     DB10.DBX 99.3;
NETWORK
TITLE = 181:
      A     #OFF;
      =     DB10.DBX 99.4;
NETWORK
TITLE = 182:
      A     #OFF;
      =     DB10.DBX 99.5;
NETWORK
TITLE = 183:
      A     #OFF;
      =     DB10.DBX 99.6;
NETWORK
TITLE = 184: press start to release the movement
      A     "F_IO".CB1_Mode_Auto;
      AN    "Error";
      AN    "DivEoff";
      AN    "ModeAuto";
      =     DB10.DBX 99.7;
NETWORK
TITLE = 185: Warning, trolley has no position
      A     "ModeAuto";
      A     "DB_ComGateway".TM.Online;
      AN    "DB_ComGateway".TM.OrderRunning;
      A(;
      L     "DB_ComGateway".TM.TroActPos;
      L     0;
      ==I;
      );
      A(;
      L     "DB_TRO"._i.ScanAreaNo;
      L     1;
      <>I;
      );
      A(;
      L     "DB_TRO"._i.ScanAreaNo;
      L     10;
      <>I;
      );
      L     S5T#10S;
      SD    T 90;
      NOP   0;
      NOP   0;
      NOP   0;
      A     T 90;
      =     DB10.DBX 98.0;
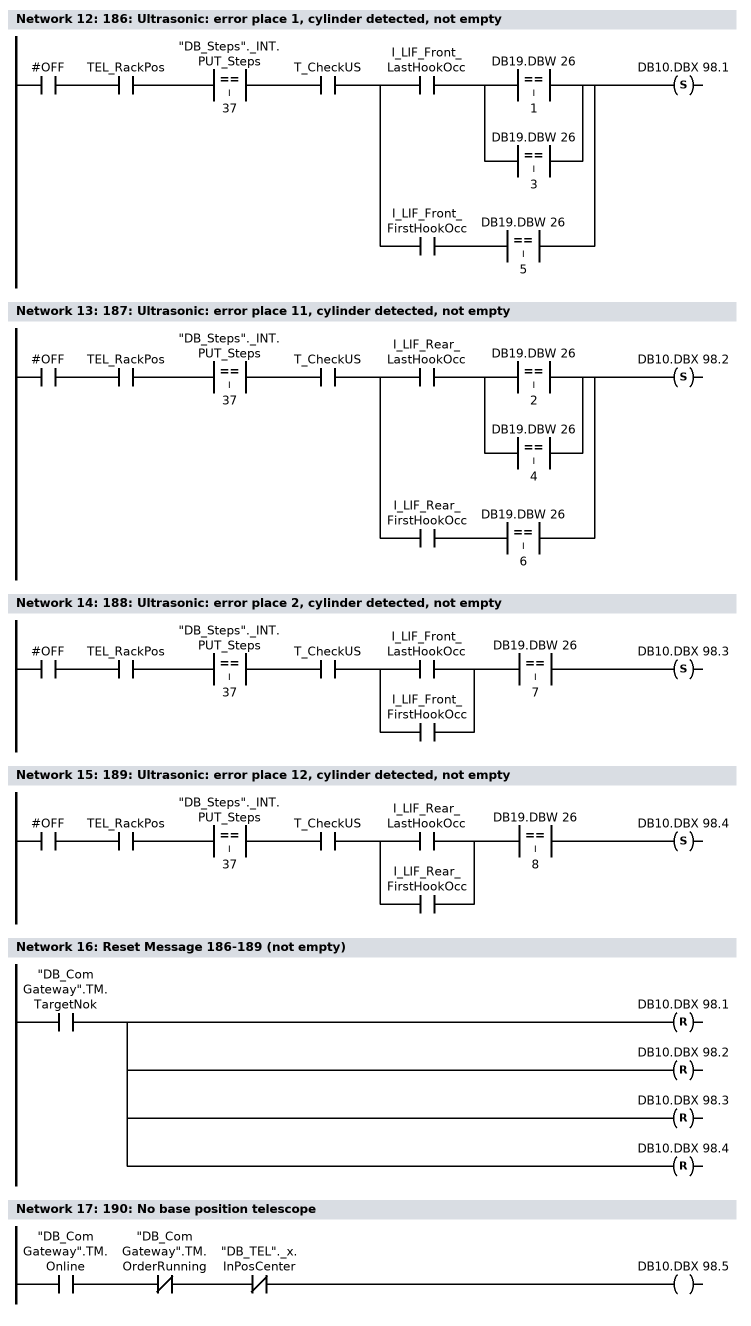
NETWORK
TITLE = 186: Ultrasonic: error place 1, cylinder detected, not empty
      A     #OFF;
      A     "TEL_RackPos";
      A(;
      L     "DB_Steps"._INT.PUT_Steps;
      L     37;
      ==I;
      );
      A     "T_CheckUS";
      A(;
      A     "I_LIF_Front_LastHookOcc";
      A(;
      O(;
      L     DB19.DBW 26;
      L     1;
      ==I;
      );
      O(;
      L     DB19.DBW 26;
      L     3;
      ==I;
      );
      );
      O;
      A     "I_LIF_Front_FirstHookOcc";
      A(;
      L     DB19.DBW 26;
      L     5;
      ==I;
      );
      );
      S     DB10.DBX 98.1;
NETWORK
TITLE = 187: Ultrasonic: error place 11, cylinder detected, not empty
      A     #OFF;
      A     "TEL_RackPos";
      A(;
      L     "DB_Steps"._INT.PUT_Steps;
      L     37;
      ==I;
      );
      A     "T_CheckUS";
      A(;
      A     "I_LIF_Rear_LastHookOcc";
      A(;
      O(;
      L     DB19.DBW 26;
      L     2;
      ==I;
      );
      O(;
      L     DB19.DBW 26;
      L     4;
      ==I;
      );
      );
      O;
      A     "I_LIF_Rear_FirstHookOcc";
      A(;
      L     DB19.DBW 26;
      L     6;
      ==I;
      );
      );
      S     DB10.DBX 98.2;
NETWORK
TITLE = 188: Ultrasonic: error place 2, cylinder detected, not empty
      A     #OFF;
      A     "TEL_RackPos";
      A(;
      L     "DB_Steps"._INT.PUT_Steps;
      L     37;
      ==I;
      );
      A     "T_CheckUS";
      A(;
      O     "I_LIF_Front_LastHookOcc";
      O     "I_LIF_Front_FirstHookOcc";
      );
      A(;
      L     DB19.DBW 26;
      L     7;
      ==I;
      );
      S     DB10.DBX 98.3;
NETWORK
TITLE = 189: Ultrasonic: error place 12, cylinder detected, not empty
      A     #OFF;
      A     "TEL_RackPos";
      A(;
      L     "DB_Steps"._INT.PUT_Steps;
      L     37;
      ==I;
      );
      A     "T_CheckUS";
      A(;
      O     "I_LIF_Rear_LastHookOcc";
      O     "I_LIF_Rear_FirstHookOcc";
      );
      A(;
      L     DB19.DBW 26;
      L     8;
      ==I;
      );
      S     DB10.DBX 98.4;
NETWORK
TITLE = Reset Message 186-189 (not empty)
      A     "DB_ComGateway".TM.TargetNok;
      R     DB10.DBX 98.1;
      R     DB10.DBX 98.2;
      R     DB10.DBX 98.3;
      R     DB10.DBX 98.4;
NETWORK
TITLE = 190: No base position telescope
      A     "DB_ComGateway".TM.Online;
      AN    "DB_ComGateway".TM.OrderRunning;
      AN    "DB_TEL"._x.InPosCenter;
      =     DB10.DBX 98.5;
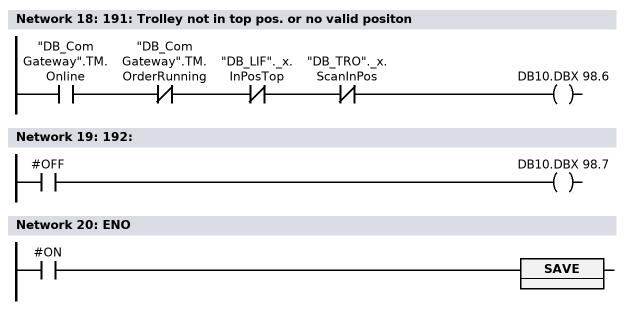
NETWORK
TITLE = 191: Trolley not in top pos. or no valid positon
      A     "DB_ComGateway".TM.Online;
      AN    "DB_ComGateway".TM.OrderRunning;
      AN    "DB_LIF"._x.InPosTop;
      AN    "DB_TRO"._x.ScanInPos;
      =     DB10.DBX 98.6;
NETWORK
TITLE = 192:
      A     #OFF;
      =     DB10.DBX 98.7;
NETWORK
TITLE = ENO
      A     #ON;
      SAVE;
END_FUNCTION

FUNCTION "CableDrum" : VOID	// FC 60
TITLE = Cable Drum
VERSION : 0.1
VAR_TEMP
  diff : INT ;
  pFl : BOOL ;
  nFl : BOOL ;
END_VAR
BEGIN
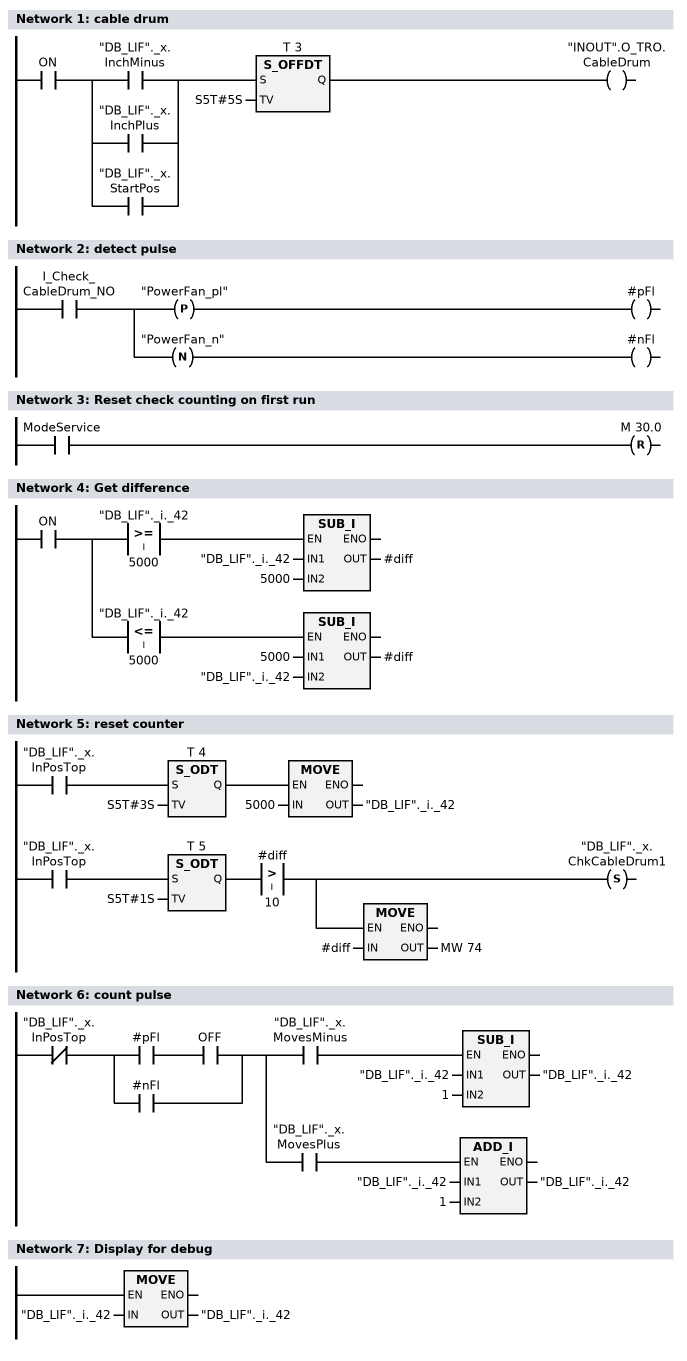
NETWORK
TITLE = cable drum
      A     "ON";
      A(;
      O     "DB_LIF"._x.InchMinus;
      O     "DB_LIF"._x.InchPlus;
      O     "DB_LIF"._x.StartPos;
      );
      L     S5T#5S;
      SF    T 3;
      NOP   0;
      NOP   0;
      NOP   0;
      A     T 3;
      =     "INOUT".O_TRO.CableDrum;
NETWORK
TITLE = detect pulse
      A     "I_Check_CableDrum_NO";
      =     L 3.0;
      A     L 3.0;
      FP    "PowerFan_pl";
      =     #pFl;
      A     L 3.0;
      FN    "PowerFan_n";
      =     #nFl;
NETWORK
TITLE = Reset check counting on first run
//after service mode the counter is sometimes off
//
      A     "ModeService";
      R     M 30.0;
NETWORK
TITLE = Get difference
      A     "ON";
      =     L 3.0;
      A     L 3.0;
      A(;
      L     "DB_LIF"._i._42;
      L     5000;
      >=I;
      );
      JNB   _001;
      L     "DB_LIF"._i._42;
      L     5000;
      -I;
      T     #diff;
_001: NOP   0;
      A     L 3.0;
      A(;
      L     "DB_LIF"._i._42;
      L     5000;
      <=I;
      );
      JNB   _002;
      L     5000;
      L     "DB_LIF"._i._42;
      -I;
      T     #diff;
_002: NOP   0;
NETWORK
TITLE = reset counter
      A     "DB_LIF"._x.InPosTop;
      =     L 3.0;
      A(;
      A     L 3.0;
      L     S5T#3S;
      SD    T 4;
      NOP   0;
      NOP   0;
      NOP   0;
      A     T 4;
      );
      JNB   _003;
      L     5000;
      T     "DB_LIF"._i._42;
_003: NOP   0;
      A(;
      A     L 3.0;
      L     S5T#1S;
      SD    T 5;
      NOP   0;
      NOP   0;
      NOP   0;
      A     T 5;
      );
      A(;
      L     #diff;
      L     10;
      >I;
      );
      =     L 3.1;
      A     L 3.1;
      BLD   102;
      S     "DB_LIF"._x.ChkCableDrum1;
      A     L 3.1;
      JNB   _004;
      L     #diff;
      T     MW 74;
_004: NOP   0;
NETWORK
TITLE = count pulse
      AN    "DB_LIF"._x.InPosTop;
      A(;
      A     #pFl;
      A     "OFF";
      O     #nFl;
      );
      =     L 3.0;
      A     L 3.0;
      A     "DB_LIF"._x.MovesMinus;
      JNB   _005;
      L     "DB_LIF"._i._42;
      L     1;
      -I;
      T     "DB_LIF"._i._42;
_005: NOP   0;
      A     L 3.0;
      A     "DB_LIF"._x.MovesPlus;
      JNB   _006;
      L     "DB_LIF"._i._42;
      L     1;
      +I;
      T     "DB_LIF"._i._42;
_006: NOP   0;
NETWORK
TITLE = Display for debug
      L     "DB_LIF"._i._42;
      T     "DB_LIF"._i._42;
      NOP   0;
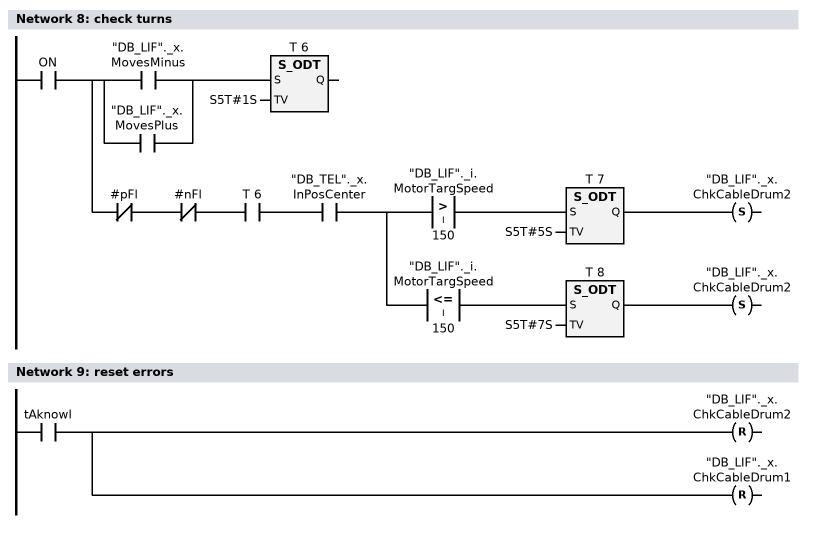
NETWORK
TITLE = check turns
      A     "ON";
      =     L 3.0;
      A     L 3.0;
      A(;
      O     "DB_LIF"._x.MovesMinus;
      O     "DB_LIF"._x.MovesPlus;
      );
      L     S5T#1S;
      SD    T 6;
      NOP   0;
      NOP   0;
      NOP   0;
      NOP   0;
      A     L 3.0;
      AN    #pFl;
      AN    #nFl;
      A     T 6;
      A     "DB_TEL"._x.InPosCenter;
      =     L 3.1;
      A     L 3.1;
      A(;
      L     "DB_LIF"._i.MotorTargSpeed;
      L     150;
      >I;
      );
      L     S5T#5S;
      SD    T 7;
      NOP   0;
      NOP   0;
      NOP   0;
      A     T 7;
      S     "DB_LIF"._x.ChkCableDrum2;
      A     L 3.1;
      A(;
      L     "DB_LIF"._i.MotorTargSpeed;
      L     150;
      <=I;
      );
      L     S5T#7S;
      SD    T 8;
      NOP   0;
      NOP   0;
      NOP   0;
      A     T 8;
      S     "DB_LIF"._x.ChkCableDrum2;
NETWORK
TITLE = reset errors
      A     "tAknowl";
      R     "DB_LIF"._x.ChkCableDrum2;
      R     "DB_LIF"._x.ChkCableDrum1;
END_FUNCTION

FUNCTION "TargetPosLift" : VOID	// FC 70
TITLE = Taget Positions Lift
//Pos Hookover
//Pos Hookunder
//Pos Teleskops
//Hook Type
//Circum Max
VERSION : 2.0
VAR_INPUT
  in_b_start : BOOL ;
  in_i_DbNo : INT ;
  in_i_DbNo_2 : INT ;
  in_LengthDataset : INT ;
  in_i_LifPosNo : INT ;
  in_i_TelPosNo : INT ;
  in_di_TelCenterpos : DINT ;
END_VAR
VAR_OUTPUT
  out_di_PosHo : DINT ;
  out_di_PosHu : DINT ;
  out_di_PosTel : DINT ;
  out_i_CircMax : INT ;
  out_i_Hooktype : INT ;
END_VAR
VAR_TEMP
  tmp_di_TelPosVal : DINT ;
  tmp_i_1 : INT ;
  tmp_i_CircumMax : INT ;
  tmp_i_HookType : INT ;
  tmp_fault : BOOL ;
  tmpRear : BOOL ;
END_VAR
BEGIN
NETWORK
TITLE = init
      L     0;
      T     #out_di_PosHo;
      T     #out_di_PosHu;
      T     #out_di_PosTel;
      T     #out_i_CircMax;
      T     #out_i_Hooktype;
      CLR;
      R     #tmp_fault;
      R     #tmpRear;
NETWORK
TITLE = start fc
      AN    #in_b_start;
      JC    flt;
NETWORK
TITLE = chk teleskopes target position
//TEL position 1..3 = "left" side DB92
//TEL position 11..13 = "right" side DB93
      A(;	// Rear side
      L     #in_i_TelPosNo;
      L     11;
      >=I;
      );
      A(;
      L     #in_i_TelPosNo;
      L     13;
      <=I;
      );
      JC    rear;
      A(;	// Front side
      L     #in_i_TelPosNo;
      L     1;
      >=I;
      );
      A(;
      L     #in_i_TelPosNo;
      L     3;
      <=I;
      );
      JC    frnt;
      JU    flt;	// no side, fault
NETWORK
TITLE =
frnt: NOP   0;
      L     #in_i_DbNo;
      T     #tmp_i_1;
      JU    nosi;
NETWORK
TITLE =
rear: NOP   0;
      L     #in_i_DbNo_2;
      T     #tmp_i_1;
      S     #tmpRear;
      JU    nosi;
NETWORK
TITLE = liftpositions
nosi: NOP   0;
      OPN   DB [#tmp_i_1];
      L     #in_i_LifPosNo;	//pointer to actual dataset
      L     1;
      -D;
      L     #in_LengthDataset;
      *D;
      A     #tmpRear;
      JCN   fr;
      L     L#560;
      +D;
fr:   SLD   3;
      LAR1;
      L     DBD [AR1,P#0.0];	//output liftpositions
      T     #out_di_PosHo;
      L     DBD [AR1,P#4.0];
      +D;
      T     #out_di_PosHu;
NETWORK
TITLE = teleskopposition
      O(;
      L     #in_i_TelPosNo;
      L     1;
      ==I;
      );
      O(;
      L     #in_i_TelPosNo;
      L     11;
      ==I;
      );
      JCN   m01;
      L     DBD [AR1,P#18.0];	//load position inside
      T     #tmp_di_TelPosVal;
      L     DBW [AR1,P#16.0];	//load position inside
      T     #tmp_i_CircumMax;
      L     DBW [AR1,P#8.0];	//load position inside
      T     #tmp_i_HookType;
      JU    m10;
m01:  NOP   0;
      O(;
      L     #in_i_TelPosNo;
      L     2;
      ==I;
      );
      O(;
      L     #in_i_TelPosNo;
      L     12;
      ==I;
      );
      JCN   m02;
      L     DBD [AR1,P#34.0];	//load position middle
      T     #tmp_di_TelPosVal;
      L     DBW [AR1,P#32.0];	//load position inside
      T     #tmp_i_CircumMax;
      L     DBW [AR1,P#24.0];	//load position inside
      T     #tmp_i_HookType;
      JU    m10;
m02:  NOP   0;
      O(;
      L     #in_i_TelPosNo;
      L     3;
      ==I;
      );
      O(;
      L     #in_i_TelPosNo;
      L     13;
      ==I;
      );
      JCN   m03;
      L     DBD [AR1,P#50.0];	//load position outside
      T     #tmp_di_TelPosVal;
      L     DBW [AR1,P#48.0];	//load position inside
      T     #tmp_i_CircumMax;
      L     DBW [AR1,P#40.0];	//load position inside
      T     #tmp_i_HookType;
      JU    m10;
m03:  L     #in_di_TelCenterpos;
m10:  NOP   0;
NETWORK
TITLE = output values
      L     #tmp_di_TelPosVal;
      T     #out_di_PosTel;
      L     #tmp_i_CircumMax;
      T     #out_i_CircMax;
      L     #tmp_i_HookType;
      T     #out_i_Hooktype;
      JU    Ende;
NETWORK
TITLE =
flt:  NOP   0;
      SET;
      S     #tmp_fault;
NETWORK
TITLE =
Ende: NOP   0;
      AN    #tmp_fault;
      SAVE;
END_FUNCTION

FUNCTION "CheckHookType" : VOID	// FC 72
TITLE = Check Hook Type
VERSION : 0.1
VAR_INPUT
  IN_HookTypeRack : INT ;
  IN_HookTypeTele : INT ;
  IN_TargetPos : DINT ;
  IN_CenterPos : DINT ;
END_VAR
VAR_OUTPUT
  OUT_HookTypeRack : BOOL ;
  OUT_HookTypeBuffer : BOOL ;
  OUT_HookTypeLS : BOOL ;
  OUT_HookTypeFaultTEL : BOOL ;
  OUT_HookTypeFaultRACK : BOOL ;
END_VAR
VAR_TEMP
  tmp_w_HookType : WORD ;
  tmp_i_ChkHookType : INT ;
  ON : BOOL ;
  tmp_HookType_101 : BOOL ;	//Zylinder
  tmp_HookType_102 : BOOL ;	//Zylinder
  tmp_HookType_103 : BOOL ;	//Zylinder
  tmp_HookType_104 : BOOL ;	//Zylinder
  tmp_HookType_105 : BOOL ;	//Zylinder
  tmp_HookType_121 : BOOL ;	//Raster
  tmp_HookType_210 : BOOL ;	//LS
  tmp_HookType_299 : BOOL ;	//RBG_Buffer
  tmp_HookType_Rack : BOOL ;
  tmp_HookType_Buffer : BOOL ;
  tmp_TelType_01 : BOOL ;	//Zylinder
  tmp_TelType_02 : BOOL ;	//Zylinder
  tmp_TelType_03 : BOOL ;	//Zylinder
  tmp_TelType_04 : BOOL ;	//Zylinder
  tmp_TelType_05 : BOOL ;	//Zylinder
  tmp_TelType_21 : BOOL ;	//LS
  tmp_TelType_99 : BOOL ;	//RBG_Buffer
  tmp_TelType_Rack : BOOL ;
  tmp_TelType_Buffer : BOOL ;
  tmp_Release : BOOL ;
END_VAR
BEGIN
